LIN {X 0,Y 251.063,Z 534.012,A -85,B 0,C 180,E1 -18793.743,E2 -18793.743} C_VEL
LIN {X 0,Y 249.355,Z 538.84,A -85,B 0,C 180,E1 -18796.138,E2 -18796.138} C_VEL
LIN {X 0,Y 248.191,Z 542.574,A -85,B 0,C 180,E1 -18798.566,E2 -18798.566} C_VEL
LIN {X 0,Y 247.654,Z 544.519,A -85,B 0,C 180,E1 -18800.195,E2 -18800.195} C_VEL
LIN {X 0,Y 247.265,Z 546.047,A -85,B 0,C 180,E1 -18801.829,E2 -18801.829} C_VEL
LIN {X 0,Y 246.923,Z 547.841,A -85,B 0,C 180,E1 -18805.101,E2 -18805.101} C_VEL
LIN {X 0,Y 246.919,Z 548.165,A -85,B 0,C 180,E1 -18806.736,E2 -18806.736} C_VEL
LIN {X 0,Y 246.996,Z 548.103,A -85,B 0,C 180,E1 -18808.368,E2 -18808.368} C_VEL
LIN {X 0,Y 247.028,Z 547.606,A -85,B 0,C 180,E1 -18809.999,E2 -18809.999} C_VEL
LIN {X 0,Y 247.019,Z 546.702,A -85,B 0,C 180,E1 -18811.629,E2 -18811.629} C_VEL
LIN {X 0,Y 246.976,Z 545.393,A -85,B 0,C 180,E1 -18813.261,E2 -18813.261} C_VEL
LIN {X 0,Y 246.983,Z 543.321,A -85,B 0,C 180,E1 -18815.163,E2 -18815.163} C_VEL
LIN {X 0,Y 247.257,Z 538.751,A -85,B 0,C 180,E1 -18818.169,E2 -18818.169} C_VEL
LIN {X 0,Y 247.724,Z 533.748,A -85,B 0,C 180,E1 -18820.625,E2 -18820.625} C_VEL
LIN {X 0,Y 248.523,Z 527.438,A -85,B 0,C 180,E1 -18823.074,E2 -18823.074} C_VEL
LIN {X 0,Y 249.77,Z 519.531,A -85,B 0,C 180,E1 -18825.503,E2 -18825.503} C_VEL
LIN {X 0,Y 251.093,Z 511.441,A -85,B 0,C 180,E1 -18827.51,E2 -18827.51} C_VEL
LIN {X 0,Y 252.671,Z 501.551,A -85,B 0,C 180,E1 -18829.497,E2 -18829.497} C_VEL
LIN {X 0,Y 253.852,Z 493.137,A -85,B 0,C 180,E1 -18830.881,E2 -18830.881} C_VEL
LIN {X 0,Y 255.388,Z 483.003,A -85,B 0,C 180,E1 -18832.232,E2 -18832.232} C_VEL
LIN {X 0,Y 256.919,Z 471.105,A -85,B 0,C 180,E1 -18833.474,E2 -18833.474} C_VEL
LIN {X 0,Y 258.118,Z 458.702,A -85,B 0,C 180,E1 -18834.425,E2 -18834.425} C_VEL
LIN {X 0,Y 259.131,Z 444.941,A -85,B 0,C 180,E1 -18835.125,E2 -18835.125} C_VEL
LIN {X 0,Y 260.839,Z 386.415,A -85,B 0,C 180,E1 -18836.75,E2 -18836.75} C_VEL
LIN {X 0,Y 257.203,Z 354.534,A -85,B 0,C 180,E1 -18838.025,E2 -18838.025} C_VEL
LIN {X 0,Y 255.532,Z 344.226,A -85,B 0,C 180,E1 -18838.495,E2 -18838.495} C_VEL
LIN {X 0,Y 252.43,Z 335.333,A -85,B 0,C 180,E1 -18839.106,E2 -18839.106} C_VEL
LIN {X 0,Y 250.392,Z 325.515,A -85,B 0,C 180,E1 -18842.644,E2 -18842.644} C_VEL
LIN {X 0,Y 249.077,Z 319.458,A -85,B 0,C 180,E1 -18844.943,E2 -18844.943} C_VEL
LIN {X 0,Y 249.022,Z 319.465,A -85,B 0,C 180,E1 -18848.379,E2 -18848.379} C_VEL
LIN {X 0,Y 248.997,Z 319.468,A -85,B 0,C 180,E1 -18852.789,E2 -18852.789} C_VEL
LIN {X 0,Y 249.014,Z 319.465,A -85,B 0,C 180,E1 -18857.362,E2 -18857.362} C_VEL
LIN {X 0,Y 249.034,Z 319.461,A -85,B 0,C 180,E1 -18861.621,E2 -18861.621} C_VEL
LIN {X 0,Y 249.055,Z 319.459,A -85,B 0,C 180,E1 -18865.641,E2 -18865.641} C_VEL
LIN {X 0,Y 249.046,Z 319.461,A -85,B 0,C 180,E1 -18869.472,E2 -18869.472} C_VEL
LIN {X 0,Y 249.067,Z 319.461,A -85,B 0,C 180,E1 -18873.162,E2 -18873.162} C_VEL
LIN {X 0,Y 249.072,Z 319.458,A -85,B 0,C 180,E1 -18876.732,E2 -18876.732} C_VEL
LIN {X 0,Y 249.103,Z 319.45,A -85,B 0,C 180,E1 -18880.211,E2 -18880.211} C_VEL
LIN {X 0,Y 249.235,Z 319.428,A -85,B 0,C 180,E1 -18883.621,E2 -18883.621} C_VEL
LIN {X 0,Y 249.245,Z 319.436,A -85,B 0,C 180,E1 -18888.616,E2 -18888.616} C_VEL
LIN {X 0,Y 249.474,Z 319.398,A -85,B 0,C 180,E1 -18891.903,E2 -18891.903} C_VEL
LIN {X 0,Y 249.428,Z 319.407,A -85,B 0,C 180,E1 -18896.77,E2 -18896.77} C_VEL
LIN {X 0,Y 249.72,Z 319.377,A -85,B 0,C 180,E1 -18900,E2 -18900} C_VEL
LIN {X 0,Y 249.425,Z 319.409,A -85,B 0,C 180,E1 -18903.231,E2 -18903.231} C_VEL
LIN {X 0,Y 249.423,Z 319.397,A -85,B 0,C 180,E1 -18906.567,E2 -18906.567} C_VEL
LIN {X 0,Y 249.336,Z 319.421,A -85,B 0,C 180,E1 -18909.737,E2 -18909.737} C_VEL
LIN {X 0,Y 249.198,Z 319.438,A -85,B 0,C 180,E1 -18914.704,E2 -18914.704} C_VEL
LIN {X 0,Y 249.132,Z 319.453,A -85,B 0,C 180,E1 -18918.078,E2 -18918.078} C_VEL
LIN {X 0,Y 249.077,Z 319.454,A -85,B 0,C 180,E1 -18921.519,E2 -18921.519} C_VEL
LIN {X 0,Y 249.111,Z 319.452,A -85,B 0,C 180,E1 -18925.476,E2 -18925.476} C_VEL
LIN {X 0,Y 249.077,Z 319.455,A -85,B 0,C 180,E1 -18928.994,E2 -18928.994} C_VEL
LIN {X 0,Y 249.025,Z 319.464,A -85,B 0,C 180,E1 -18932.427,E2 -18932.427} C_VEL
LIN {X 0,Y 249.041,Z 319.462,A -85,B 0,C 180,E1 -18936.344,E2 -18936.344} C_VEL
LIN {X 0,Y 248.973,Z 319.469,A -85,B 0,C 180,E1 -18940.485,E2 -18940.485} C_VEL
LIN {X 0,Y 248.957,Z 319.471,A -85,B 0,C 180,E1 -18944.89,E2 -18944.89} C_VEL
LIN {X 0,Y 248.975,Z 319.469,A -85,B 0,C 180,E1 -18947.356,E2 -18947.356} C_VEL
LIN {X 0,Y 249.038,Z 319.461,A -85,B 0,C 180,E1 -18952.203,E2 -18952.203} C_VEL
LIN {X 0,Y 249.04,Z 319.462,A -85,B 0,C 180,E1 -18955.641,E2 -18955.641} C_VEL
LIN {X 0,Y 249,Z 319.468,A -85,B 0,C 180,E1 -18959.468,E2 -18959.468} C_VEL
LIN {X 0,Y 249.033,Z 319.465,A -85,B 0,C 180,E1 -18963.159,E2 -18963.159} C_VEL
LIN {X 0,Y 249.053,Z 319.461,A -85,B 0,C 180,E1 -18966.732,E2 -18966.732} C_VEL
LIN {X 0,Y 249.085,Z 319.458,A -85,B 0,C 180,E1 -18970.211,E2 -18970.211} C_VEL
LIN {X 0,Y 249.248,Z 319.437,A -85,B 0,C 180,E1 -18974.695,E2 -18974.695} C_VEL
LIN {X 0,Y 250.36,Z 322.47,A -85,B 0,C 180,E1 -18974.92,E2 -18974.92} C_VEL
LIN {X 0,Y 255.478,Z 334.885,A -85,B 0,C 180,E1 -18975.815,E2 -18975.815} C_VEL
LIN {X 0,Y 261.05,Z 350.896,A -85,B 0,C 180,E1 -18976.822,E2 -18976.822} C_VEL
LIN {X 0,Y 261.764,Z 354.425,A -85,B 0,C 180,E1 -18976.99,E2 -18976.99} C_VEL
LIN {X 0,Y 259.347,Z 426.547,A -85,B 0,C 180,E1 -18978.948,E2 -18978.948} C_VEL
LIN {X 0,Y 258.556,Z 440.569,A -85,B 0,C 180,E1 -18979.676,E2 -18979.676} C_VEL
LIN {X 0,Y 257.383,Z 453.393,A -85,B 0,C 180,E1 -18980.671,E2 -18980.671} C_VEL
LIN {X 0,Y 256.154,Z 465.078,A -85,B 0,C 180,E1 -18981.918,E2 -18981.918} C_VEL
LIN {X 0,Y 254.644,Z 476.639,A -85,B 0,C 180,E1 -18983.505,E2 -18983.505} C_VEL
LIN {X 0,Y 253.095,Z 486.581,A -85,B 0,C 180,E1 -18985.223,E2 -18985.223} C_VEL
LIN {X 0,Y 251.502,Z 495.769,A -85,B 0,C 180,E1 -18987.198,E2 -18987.198} C_VEL
LIN {X 0,Y 250.012,Z 504.701,A -85,B 0,C 180,E1 -18989.599,E2 -18989.599} C_VEL
LIN {X 0,Y 248.864,Z 511.881,A -85,B 0,C 180,E1 -18992.024,E2 -18992.024} C_VEL
LIN {X 0,Y 247.927,Z 518.411,A -85,B 0,C 180,E1 -18994.88,E2 -18994.88} C_VEL
LIN {X 0,Y 247.376,Z 522.735,A -85,B 0,C 180,E1 -18997.346,E2 -18997.346} C_VEL
LIN {X 0,Y 246.917,Z 525.994,A -85,B 0,C 180,E1 -18999.834,E2 -18999.834} C_VEL
LIN {X 0,Y 246.776,Z 527.616,A -85,B 0,C 180,E1 -19001.5,E2 -19001.5} C_VEL
LIN {X 0,Y 246.791,Z 529.434,A -85,B 0,C 180,E1 -19004.479,E2 -19004.479} C_VEL
LIN {X 0,Y 246.83,Z 529.9,A -85,B 0,C 180,E1 -19006.544,E2 -19006.544} C_VEL
LIN {X 0,Y 247.068,Z 529.849,A -85,B 0,C 180,E1 -19008.235,E2 -19008.235} C_VEL
LIN {X 0,Y 247.581,Z 529.079,A -85,B 0,C 180,E1 -19010.485,E2 -19010.485} C_VEL
LIN {X 0,Y 248.484,Z 527.059,A -85,B 0,C 180,E1 -19013.327,E2 -19013.327} C_VEL
LIN {X 0,Y 249.626,Z 524.337,A -85,B 0,C 180,E1 -19015.719,E2 -19015.719} C_VEL
LIN {X 0,Y 251.27,Z 520.117,A -85,B 0,C 180,E1 -19018.392,E2 -19018.392} C_VEL
LIN {X 0,Y 253.306,Z 514.524,A -85,B 0,C 180,E1 -19021.018,E2 -19021.018} C_VEL
LIN {X 0,Y 255.581,Z 508.057,A -85,B 0,C 180,E1 -19023.365,E2 -19023.365} C_VEL
LIN {X 0,Y 258.262,Z 499.864,A -85,B 0,C 180,E1 -19025.713,E2 -19025.713} C_VEL
LIN {X 0,Y 261.05,Z 490.753,A -85,B 0,C 180,E1 -19027.77,E2 -19027.77} C_VEL
LIN {X 0,Y 264.031,Z 479.746,A -85,B 0,C 180,E1 -19029.706,E2 -19029.706} C_VEL
LIN {X 0,Y 266.539,Z 468.701,A -85,B 0,C 180,E1 -19031.239,E2 -19031.239} C_VEL
LIN {X 0,Y 268.671,Z 457.188,A -85,B 0,C 180,E1 -19032.471,E2 -19032.471} C_VEL
LIN {X 0,Y 270.514,Z 444.524,A -85,B 0,C 180,E1 -19033.482,E2 -19033.482} C_VEL
LIN {X 0,Y 271.823,Z 431.405,A -85,B 0,C 180,E1 -19034.215,E2 -19034.215} C_VEL
LIN {X 0,Y 272.675,Z 416.434,A -85,B 0,C 180,E1 -19034.695,E2 -19034.695} C_VEL
LIN {X 0,Y 274.89,Z 366.849,A -85,B 0,C 180,E1 -19035.961,E2 -19035.961} C_VEL
LIN {X 0,Y 268.89,Z 353.904,A -85,B 0,C 180,E1 -19037.381,E2 -19037.381} C_VEL
LIN {X 0,Y 260.051,Z 337.508,A -85,B 0,C 180,E1 -19039.563,E2 -19039.563} C_VEL
LIN {X 0,Y 253.907,Z 327.715,A -85,B 0,C 180,E1 -19041.162,E2 -19041.162} C_VEL
LIN {X 0,Y 251.471,Z 323.932,A -85,B 0,C 180,E1 -19041.827,E2 -19041.827} C_VEL
LIN {X 0,Y 249.688,Z 321.608,A -85,B 0,C 180,E1 -19042.308,E2 -19042.308} C_VEL
LIN {X 0,Y 249.177,Z 320.079,A -85,B 0,C 180,E1 -19042.516,E2 -19042.516} C_VEL
LIN {X 0,Y 249.108,Z 319.459,A -85,B 0,C 180,E1 -19042.838,E2 -19042.838} C_VEL
LIN {X 0,Y 249.034,Z 319.461,A -85,B 0,C 180,E1 -19047.574,E2 -19047.574} C_VEL
LIN {X 0,Y 249.1,Z 319.457,A -85,B 0,C 180,E1 -19051.338,E2 -19051.338} C_VEL
LIN {X 0,Y 249.154,Z 319.45,A -85,B 0,C 180,E1 -19054.969,E2 -19054.969} C_VEL
LIN {X 0,Y 249.113,Z 319.446,A -85,B 0,C 180,E1 -19060.212,E2 -19060.212} C_VEL
LIN {X 0,Y 249.245,Z 319.437,A -85,B 0,C 180,E1 -19063.622,E2 -19063.622} C_VEL
LIN {X 0,Y 249.255,Z 319.436,A -85,B 0,C 180,E1 -19068.617,E2 -19068.617} C_VEL
LIN {X 0,Y 249.484,Z 319.4,A -85,B 0,C 180,E1 -19071.903,E2 -19071.903} C_VEL
LIN {X 0,Y 249.435,Z 319.403,A -85,B 0,C 180,E1 -19076.769,E2 -19076.769} C_VEL
LIN {X 0,Y 249.723,Z 319.363,A -85,B 0,C 180,E1 -19080,E2 -19080} C_VEL
LIN {X 0,Y 249.437,Z 319.41,A -85,B 0,C 180,E1 -19083.23,E2 -19083.23} C_VEL
LIN {X 0,Y 249.445,Z 319.395,A -85,B 0,C 180,E1 -19086.358,E2 -19086.358} C_VEL
LIN {X 0,Y 248.906,Z 319.472,A -85,B 0,C 180,E1 -19087.704,E2 -19087.704} C_VEL
LIN {X 0,Y 247.33,Z 319.675,A -85,B 0,C 180,E1 -19089.024,E2 -19089.024} C_VEL
LIN {X 0,Y 243.425,Z 320.169,A -85,B 0,C 180,E1 -19091.678,E2 -19091.678} C_VEL
LIN {X 0,Y 242.273,Z 320.307,A -85,B 0,C 180,E1 -19093.067,E2 -19093.067} C_VEL
LIN {X 0,Y 242.162,Z 320.316,A -85,B 0,C 180,E1 -19093.539,E2 -19093.539} C_VEL
LIN {X 0,Y 242.153,Z 320.307,A -85,B 0,C 180,E1 -19096.872,E2 -19096.872} C_VEL
LIN {X 0,Y 242.029,Z 320.324,A -85,B 0,C 180,E1 -19101.686,E2 -19101.686} C_VEL
LIN {X 0,Y 242.069,Z 320.318,A -85,B 0,C 180,E1 -19105.838,E2 -19105.838} C_VEL
LIN {X 0,Y 242.033,Z 320.324,A -85,B 0,C 180,E1 -19109.58,E2 -19109.58} C_VEL
LIN {X 0,Y 241.983,Z 320.332,A -85,B 0,C 180,E1 -19113.492,E2 -19113.492} C_VEL
LIN {X 0,Y 241.992,Z 320.333,A -85,B 0,C 180,E1 -19117.582,E2 -19117.582} C_VEL
LIN {X 0,Y 241.936,Z 320.351,A -85,B 0,C 180,E1 -19121.923,E2 -19121.923} C_VEL
LIN {X 0,Y 241.936,Z 320.499,A -85,B 0,C 180,E1 -19124.086,E2 -19124.086} C_VEL
LIN {X 0,Y 244.233,Z 327.949,A -85,B 0,C 180,E1 -19128.121,E2 -19128.121} C_VEL
LIN {X 0,Y 245.847,Z 333.529,A -85,B 0,C 180,E1 -19130.843,E2 -19130.843} C_VEL
LIN {X 0,Y 248.328,Z 337.884,A -85,B 0,C 180,E1 -19131.574,E2 -19131.574} C_VEL
LIN {X 0,Y 254.341,Z 348.606,A -85,B 0,C 180,E1 -19133.258,E2 -19133.258} C_VEL
LIN {X 0,Y 261.31,Z 362.634,A -85,B 0,C 180,E1 -19135.116,E2 -19135.116} C_VEL
LIN {X 0,Y 265.318,Z 371.754,A -85,B 0,C 180,E1 -19136.15,E2 -19136.15} C_VEL
LIN {X 0,Y 268.268,Z 390.386,A -85,B 0,C 180,E1 -19137.283,E2 -19137.283} C_VEL
LIN {X 0,Y 265.892,Z 443.094,A -85,B 0,C 180,E1 -19138.704,E2 -19138.704} C_VEL
LIN {X 0,Y 264.543,Z 456.576,A -85,B 0,C 180,E1 -19139.333,E2 -19139.333} C_VEL
LIN {X 0,Y 262.561,Z 469.325,A -85,B 0,C 180,E1 -19140.206,E2 -19140.206} C_VEL
LIN {X 0,Y 260.161,Z 481.261,A -85,B 0,C 180,E1 -19141.346,E2 -19141.346} C_VEL
LIN {X 0,Y 257.375,Z 492.686,A -85,B 0,C 180,E1 -19142.781,E2 -19142.781} C_VEL
LIN {X 0,Y 254.574,Z 502.997,A -85,B 0,C 180,E1 -19144.445,E2 -19144.445} C_VEL
LIN {X 0,Y 251.89,Z 511.459,A -85,B 0,C 180,E1 -19146.135,E2 -19146.135} C_VEL
LIN {X 0,Y 248.808,Z 520.659,A -85,B 0,C 180,E1 -19148.456,E2 -19148.456} C_VEL
LIN {X 0,Y 246.34,Z 528.074,A -85,B 0,C 180,E1 -19150.846,E2 -19150.846} C_VEL
LIN {X 0,Y 244.26,Z 534.062,A -85,B 0,C 180,E1 -19153.277,E2 -19153.277} C_VEL
LIN {X 0,Y 242.433,Z 538.823,A -85,B 0,C 180,E1 -19155.734,E2 -19155.734} C_VEL
LIN {X 0,Y 241.217,Z 542.494,A -85,B 0,C 180,E1 -19158.231,E2 -19158.231} C_VEL
LIN {X 0,Y 240.641,Z 544.408,A -85,B 0,C 180,E1 -19159.907,E2 -19159.907} C_VEL
LIN {X 0,Y 240.215,Z 545.881,A -85,B 0,C 180,E1 -19161.587,E2 -19161.587} C_VEL
LIN {X 0,Y 239.845,Z 547.617,A -85,B 0,C 180,E1 -19164.956,E2 -19164.956} C_VEL
LIN {X 0,Y 239.821,Z 547.913,A -85,B 0,C 180,E1 -19166.639,E2 -19166.639} C_VEL
LIN {X 0,Y 239.902,Z 547.807,A -85,B 0,C 180,E1 -19168.32,E2 -19168.32} C_VEL
LIN {X 0,Y 239.957,Z 547.272,A -85,B 0,C 180,E1 -19169.999,E2 -19169.999} C_VEL
LIN {X 0,Y 239.949,Z 546.34,A -85,B 0,C 180,E1 -19171.677,E2 -19171.677} C_VEL
LIN {X 0,Y 239.876,Z 545,A -85,B 0,C 180,E1 -19173.358,E2 -19173.358} C_VEL
LIN {X 0,Y 239.919,Z 542.144,A -85,B 0,C 180,E1 -19175.883,E2 -19175.883} C_VEL
LIN {X 0,Y 240.197,Z 538.234,A -85,B 0,C 180,E1 -19178.411,E2 -19178.411} C_VEL
LIN {X 0,Y 240.703,Z 533.162,A -85,B 0,C 180,E1 -19180.939,E2 -19180.939} C_VEL
LIN {X 0,Y 241.577,Z 526.769,A -85,B 0,C 180,E1 -19183.457,E2 -19183.457} C_VEL
LIN {X 0,Y 242.873,Z 518.738,A -85,B 0,C 180,E1 -19185.955,E2 -19185.955} C_VEL
LIN {X 0,Y 244.141,Z 511.311,A -85,B 0,C 180,E1 -19187.841,E2 -19187.841} C_VEL
LIN {X 0,Y 245.738,Z 501.719,A -85,B 0,C 180,E1 -19189.83,E2 -19189.83} C_VEL
LIN {X 0,Y 246.977,Z 493.264,A -85,B 0,C 180,E1 -19191.272,E2 -19191.272} C_VEL
LIN {X 0,Y 248.785,Z 481.618,A -85,B 0,C 180,E1 -19192.855,E2 -19192.855} C_VEL
LIN {X 0,Y 250.355,Z 469.287,A -85,B 0,C 180,E1 -19194.128,E2 -19194.128} C_VEL
LIN {X 0,Y 251.652,Z 456.296,A -85,B 0,C 180,E1 -19195.095,E2 -19195.095} C_VEL
LIN {X 0,Y 252.543,Z 443.755,A -85,B 0,C 180,E1 -19195.717,E2 -19195.717} C_VEL
LIN {X 0,Y 254.155,Z 384.923,A -85,B 0,C 180,E1 -19197.39,E2 -19197.39} C_VEL
LIN {X 0,Y 249.791,Z 349.447,A -85,B 0,C 180,E1 -19198.899,E2 -19198.899} C_VEL
LIN {X 0,Y 248.836,Z 345.277,A -85,B 0,C 180,E1 -19199.125,E2 -19199.125} C_VEL
LIN {X 0,Y 245.191,Z 335.113,A -85,B 0,C 180,E1 -19199.838,E2 -19199.838} C_VEL
LIN {X 0,Y 242.941,Z 324.443,A -85,B 0,C 180,E1 -19203.838,E2 -19203.838} C_VEL
LIN {X 0,Y 242.001,Z 320.339,A -85,B 0,C 180,E1 -19205.506,E2 -19205.506} C_VEL
LIN {X 0,Y 241.953,Z 320.343,A -85,B 0,C 180,E1 -19209.718,E2 -19209.718} C_VEL
LIN {X 0,Y 241.919,Z 320.351,A -85,B 0,C 180,E1 -19214.202,E2 -19214.202} C_VEL
LIN {X 0,Y 241.94,Z 320.348,A -85,B 0,C 180,E1 -19218.078,E2 -19218.078} C_VEL
LIN {X 0,Y 241.998,Z 320.34,A -85,B 0,C 180,E1 -19222.42,E2 -19222.42} C_VEL
LIN {X 0,Y 241.985,Z 320.342,A -85,B 0,C 180,E1 -19226.508,E2 -19226.508} C_VEL
LIN {X 0,Y 242.031,Z 320.336,A -85,B 0,C 180,E1 -19230.586,E2 -19230.586} C_VEL
LIN {X 0,Y 242.061,Z 320.33,A -85,B 0,C 180,E1 -19234.182,E2 -19234.182} C_VEL
LIN {X 0,Y 242.046,Z 320.333,A -85,B 0,C 180,E1 -19238.297,E2 -19238.297} C_VEL
LIN {X 0,Y 242.156,Z 320.306,A -85,B 0,C 180,E1 -19243.278,E2 -19243.278} C_VEL
LIN {X 0,Y 242.178,Z 320.316,A -85,B 0,C 180,E1 -19248.279,E2 -19248.279} C_VEL
LIN {X 0,Y 242.42,Z 320.278,A -85,B 0,C 180,E1 -19251.665,E2 -19251.665} C_VEL
LIN {X 0,Y 242.251,Z 320.291,A -85,B 0,C 180,E1 -19255.007,E2 -19255.007} C_VEL
LIN {X 0,Y 242.629,Z 320.259,A -85,B 0,C 180,E1 -19258.34,E2 -19258.34} C_VEL
LIN {X 0,Y 242.628,Z 320.26,A -85,B 0,C 180,E1 -19261.66,E2 -19261.66} C_VEL
LIN {X 0,Y 242.4,Z 320.271,A -85,B 0,C 180,E1 -19266.66,E2 -19266.66} C_VEL
LIN {X 0,Y 242.26,Z 320.304,A -85,B 0,C 180,E1 -19270.024,E2 -19270.024} C_VEL
LIN {X 0,Y 242.16,Z 320.314,A -85,B 0,C 180,E1 -19275.141,E2 -19275.141} C_VEL
LIN {X 0,Y 242.066,Z 320.331,A -85,B 0,C 180,E1 -19278.625,E2 -19278.625} C_VEL
LIN {X 0,Y 242,Z 320.337,A -85,B 0,C 180,E1 -19282.181,E2 -19282.181} C_VEL
LIN {X 0,Y 242.061,Z 320.331,A -85,B 0,C 180,E1 -19285.839,E2 -19285.839} C_VEL
LIN {X 0,Y 242.025,Z 320.333,A -85,B 0,C 180,E1 -19289.581,E2 -19289.581} C_VEL
LIN {X 0,Y 241.975,Z 320.336,A -85,B 0,C 180,E1 -19293.494,E2 -19293.494} C_VEL
LIN {X 0,Y 241.982,Z 320.338,A -85,B 0,C 180,E1 -19297.584,E2 -19297.584} C_VEL
LIN {X 0,Y 241.903,Z 320.349,A -85,B 0,C 180,E1 -19301.93,E2 -19301.93} C_VEL
LIN {X 0,Y 241.896,Z 320.353,A -85,B 0,C 180,E1 -19306.581,E2 -19306.581} C_VEL
LIN {X 0,Y 241.989,Z 320.34,A -85,B 0,C 180,E1 -19311.643,E2 -19311.643} C_VEL
LIN {X 0,Y 241.977,Z 320.342,A -85,B 0,C 180,E1 -19314.489,E2 -19314.489} C_VEL
LIN {X 0,Y 241.95,Z 320.345,A -85,B 0,C 180,E1 -19318.478,E2 -19318.478} C_VEL
LIN {X 0,Y 241.966,Z 320.343,A -85,B 0,C 180,E1 -19322.309,E2 -19322.309} C_VEL
LIN {X 0,Y 242.023,Z 320.337,A -85,B 0,C 180,E1 -19326.014,E2 -19326.014} C_VEL
LIN {X 0,Y 242.02,Z 320.336,A -85,B 0,C 180,E1 -19329.608,E2 -19329.608} C_VEL
LIN {X 0,Y 242.165,Z 320.397,A -85,B 0,C 180,E1 -19333.974,E2 -19333.974} C_VEL
LIN {X 0,Y 243.252,Z 323.281,A -85,B 0,C 180,E1 -19334.187,E2 -19334.187} C_VEL
LIN {X 0,Y 247.71,Z 333.288,A -85,B 0,C 180,E1 -19334.983,E2 -19334.983} C_VEL
LIN {X 0,Y 254.637,Z 352.807,A -85,B 0,C 180,E1 -19336.279,E2 -19336.279} C_VEL
LIN {X 0,Y 255.173,Z 355.269,A -85,B 0,C 180,E1 -19336.405,E2 -19336.405} C_VEL
LIN {X 0,Y 252.769,Z 426.097,A -85,B 0,C 180,E1 -19338.367,E2 -19338.367} C_VEL
LIN {X 0,Y 251.992,Z 439.389,A -85,B 0,C 180,E1 -19339.049,E2 -19339.049} C_VEL
LIN {X 0,Y 250.825,Z 452.119,A -85,B 0,C 180,E1 -19340.017,E2 -19340.017} C_VEL
LIN {X 0,Y 249.515,Z 464.201,A -85,B 0,C 180,E1 -19341.293,E2 -19341.293} C_VEL
LIN {X 0,Y 248.126,Z 474.723,A -85,B 0,C 180,E1 -19342.728,E2 -19342.728} C_VEL
LIN {X 0,Y 246.484,Z 485.026,A -85,B 0,C 180,E1 -19344.479,E2 -19344.479} C_VEL
LIN {X 0,Y 245.015,Z 493.699,A -85,B 0,C 180,E1 -19346.301,E2 -19346.301} C_VEL
LIN {X 0,Y 243.608,Z 501.688,A -85,B 0,C 180,E1 -19348.348,E2 -19348.348} C_VEL
LIN {X 0,Y 242.236,Z 509.503,A -85,B 0,C 180,E1 -19350.832,E2 -19350.832} C_VEL
LIN {X 0,Y 241.248,Z 515.75,A -85,B 0,C 180,E1 -19353.341,E2 -19353.341} C_VEL
LIN {X 0,Y 240.629,Z 520.473,A -85,B 0,C 180,E1 -19355.728,E2 -19355.728} C_VEL
LIN {X 0,Y 240.057,Z 524.561,A -85,B 0,C 180,E1 -19358.418,E2 -19358.418} C_VEL
LIN {X 0,Y 239.798,Z 526.552,A -85,B 0,C 180,E1 -19360.129,E2 -19360.129} C_VEL
LIN {X 0,Y 239.681,Z 528.111,A -85,B 0,C 180,E1 -19361.846,E2 -19361.846} C_VEL
LIN {X 0,Y 239.713,Z 529.702,A -85,B 0,C 180,E1 -19364.644,E2 -19364.644} C_VEL
LIN {X 0,Y 239.783,Z 530.199,A -85,B 0,C 180,E1 -19367.045,E2 -19367.045} C_VEL
LIN {X 0,Y 240.07,Z 530.059,A -85,B 0,C 180,E1 -19368.786,E2 -19368.786} C_VEL
LIN {X 0,Y 240.571,Z 529.358,A -85,B 0,C 180,E1 -19370.796,E2 -19370.796} C_VEL
LIN {X 0,Y 241.666,Z 527.077,A -85,B 0,C 180,E1 -19374.026,E2 -19374.026} C_VEL
LIN {X 0,Y 242.767,Z 524.638,A -85,B 0,C 180,E1 -19376.176,E2 -19376.176} C_VEL
LIN {X 0,Y 244.7,Z 519.876,A -85,B 0,C 180,E1 -19379.227,E2 -19379.227} C_VEL
LIN {X 0,Y 247.211,Z 513.382,A -85,B 0,C 180,E1 -19382.212,E2 -19382.212} C_VEL
LIN {X 0,Y 249.795,Z 506.389,A -85,B 0,C 180,E1 -19384.672,E2 -19384.672} C_VEL
LIN {X 0,Y 252.323,Z 498.812,A -85,B 0,C 180,E1 -19386.788,E2 -19386.788} C_VEL
LIN {X 0,Y 255.489,Z 488.727,A -85,B 0,C 180,E1 -19388.995,E2 -19388.995} C_VEL
LIN {X 0,Y 258.373,Z 478.487,A -85,B 0,C 180,E1 -19390.756,E2 -19390.756} C_VEL
LIN {X 0,Y 260.973,Z 466.927,A -85,B 0,C 180,E1 -19392.319,E2 -19392.319} C_VEL
LIN {X 0,Y 263.246,Z 454.87,A -85,B 0,C 180,E1 -19393.562,E2 -19393.562} C_VEL
LIN {X 0,Y 265.009,Z 442.377,A -85,B 0,C 180,E1 -19394.517,E2 -19394.517} C_VEL
LIN {X 0,Y 266.236,Z 429.336,A -85,B 0,C 180,E1 -19395.192,E2 -19395.192} C_VEL
LIN {X 0,Y 267.289,Z 411.227,A -85,B 0,C 180,E1 -19395.715,E2 -19395.715} C_VEL
LIN {X 0,Y 269.108,Z 368.812,A -85,B 0,C 180,E1 -19396.84,E2 -19396.84} C_VEL
LIN {X 0,Y 262.767,Z 355.414,A -85,B 0,C 180,E1 -19398.411,E2 -19398.411} C_VEL
LIN {X 0,Y 255.455,Z 341.823,A -85,B 0,C 180,E1 -19400.309,E2 -19400.309} C_VEL
LIN {X 0,Y 249.505,Z 332.272,A -85,B 0,C 180,E1 -19401.926,E2 -19401.926} C_VEL
LIN {X 0,Y 247.267,Z 328.916,A -85,B 0,C 180,E1 -19402.556,E2 -19402.556} C_VEL
LIN {X 0,Y 245.28,Z 325.85,A -85,B 0,C 180,E1 -19403.136,E2 -19403.136} C_VEL
LIN {X 0,Y 244.295,Z 324.728,A -85,B 0,C 180,E1 -19403.413,E2 -19403.413} C_VEL
LIN {X 0,Y 242.626,Z 322.509,A -85,B 0,C 180,E1 -19403.904,E2 -19403.904} C_VEL
LIN {X 0,Y 242.017,Z 320.466,A -85,B 0,C 180,E1 -19404.175,E2 -19404.175} C_VEL
LIN {X 0,Y 241.978,Z 320.345,A -85,B 0,C 180,E1 -19408.48,E2 -19408.48} C_VEL
LIN {X 0,Y 242.012,Z 320.335,A -85,B 0,C 180,E1 -19412.313,E2 -19412.313} C_VEL
LIN {X 0,Y 242.06,Z 320.327,A -85,B 0,C 180,E1 -19416.016,E2 -19416.016} C_VEL
LIN {X 0,Y 242.04,Z 320.332,A -85,B 0,C 180,E1 -19419.608,E2 -19419.608} C_VEL
LIN {X 0,Y 242.166,Z 320.32,A -85,B 0,C 180,E1 -19423.278,E2 -19423.278} C_VEL
LIN {X 0,Y 242.189,Z 320.316,A -85,B 0,C 180,E1 -19428.28,E2 -19428.28} C_VEL
LIN {X 0,Y 242.43,Z 320.276,A -85,B 0,C 180,E1 -19431.666,E2 -19431.666} C_VEL
LIN {X 0,Y 242.259,Z 320.294,A -85,B 0,C 180,E1 -19435.007,E2 -19435.007} C_VEL
LIN {X 0,Y 242.637,Z 320.26,A -85,B 0,C 180,E1 -19438.34,E2 -19438.34} C_VEL
LIN {X 0,Y 242.638,Z 320.243,A -85,B 0,C 180,E1 -19441.66,E2 -19441.66} C_VEL
LIN {X 0,Y 242.436,Z 320.269,A -85,B 0,C 180,E1 -19446.659,E2 -19446.659} C_VEL
LIN {X 0,Y 242.348,Z 320.284,A -85,B 0,C 180,E1 -19450.02,E2 -19450.02} C_VEL
LIN {X 0,Y 242.162,Z 320.316,A -85,B 0,C 180,E1 -19453.539,E2 -19453.539} C_VEL
LIN {X 0,Y 241.428,Z 320.404,A -85,B 0,C 180,E1 -19454.926,E2 -19454.926} C_VEL
LIN {X 0,Y 238.489,Z 320.765,A -85,B 0,C 180,E1 -19457.186,E2 -19457.186} C_VEL
LIN {X 0,Y 236.053,Z 321.08,A -85,B 0,C 180,E1 -19459.028,E2 -19459.028} C_VEL
LIN {X 0,Y 235.054,Z 321.193,A -85,B 0,C 180,E1 -19460.459,E2 -19460.459} C_VEL
LIN {X 0,Y 234.996,Z 321.198,A -85,B 0,C 180,E1 -19460.944,E2 -19460.944} C_VEL
LIN {X 0,Y 234.997,Z 321.2,A -85,B 0,C 180,E1 -19466.206,E2 -19466.206} C_VEL
LIN {X 0,Y 234.934,Z 321.209,A -85,B 0,C 180,E1 -19470.567,E2 -19470.567} C_VEL
LIN {X 0,Y 234.933,Z 321.212,A -85,B 0,C 180,E1 -19474.638,E2 -19474.638} C_VEL
LIN {X 0,Y 234.944,Z 321.22,A -85,B 0,C 180,E1 -19478.944,E2 -19478.944} C_VEL
LIN {X 0,Y 234.909,Z 321.433,A -85,B 0,C 180,E1 -19482.577,E2 -19482.577} C_VEL
LIN {X 0,Y 237.376,Z 329.255,A -85,B 0,C 180,E1 -19487.08,E2 -19487.08} C_VEL
LIN {X 0,Y 238.5,Z 333.251,A -85,B 0,C 180,E1 -19489.071,E2 -19489.071} C_VEL
LIN {X 0,Y 241.379,Z 338,A -85,B 0,C 180,E1 -19489.983,E2 -19489.983} C_VEL
LIN {X 0,Y 247.642,Z 348.829,A -85,B 0,C 180,E1 -19491.858,E2 -19491.858} C_VEL
LIN {X 0,Y 255.057,Z 363.424,A -85,B 0,C 180,E1 -19493.955,E2 -19493.955} C_VEL
LIN {X 0,Y 259.996,Z 374.477,A -85,B 0,C 180,E1 -19495.296,E2 -19495.296} C_VEL
LIN {X 0,Y 262.692,Z 391.848,A -85,B 0,C 180,E1 -19496.389,E2 -19496.389} C_VEL
LIN {X 0,Y 260.18,Z 443.362,A -85,B 0,C 180,E1 -19497.797,E2 -19497.797} C_VEL
LIN {X 0,Y 258.682,Z 457.433,A -85,B 0,C 180,E1 -19498.479,E2 -19498.479} C_VEL
LIN {X 0,Y 256.674,Z 469.553,A -85,B 0,C 180,E1 -19499.337,E2 -19499.337} C_VEL
LIN {X 0,Y 254.002,Z 482.139,A -85,B 0,C 180,E1 -19500.585,E2 -19500.585} C_VEL
LIN {X 0,Y 251.123,Z 493.356,A -85,B 0,C 180,E1 -19502.045,E2 -19502.045} C_VEL
LIN {X 0,Y 248.228,Z 503.49,A -85,B 0,C 180,E1 -19503.743,E2 -19503.743} C_VEL
LIN {X 0,Y 245.44,Z 511.823,A -85,B 0,C 180,E1 -19505.467,E2 -19505.467} C_VEL
LIN {X 0,Y 242.209,Z 520.886,A -85,B 0,C 180,E1 -19507.838,E2 -19507.838} C_VEL
LIN {X 0,Y 239.642,Z 528.212,A -85,B 0,C 180,E1 -19510.289,E2 -19510.289} C_VEL
LIN {X 0,Y 237.457,Z 534.119,A -85,B 0,C 180,E1 -19512.783,E2 -19512.783} C_VEL
LIN {X 0,Y 235.534,Z 538.808,A -85,B 0,C 180,E1 -19515.307,E2 -19515.307} C_VEL
LIN {X 0,Y 234.254,Z 542.414,A -85,B 0,C 180,E1 -19517.876,E2 -19517.876} C_VEL
LIN {X 0,Y 233.615,Z 544.29,A -85,B 0,C 180,E1 -19519.6,E2 -19519.6} C_VEL
LIN {X 0,Y 232.89,Z 546.744,A -85,B 0,C 180,E1 -19523.066,E2 -19523.066} C_VEL
LIN {X 0,Y 232.761,Z 547.491,A -85,B 0,C 180,E1 -19525.14,E2 -19525.14} C_VEL
LIN {X 0,Y 232.811,Z 547.499,A -85,B 0,C 180,E1 -19528.269,E2 -19528.269} C_VEL
LIN {X 0,Y 232.888,Z 546.938,A -85,B 0,C 180,E1 -19529.999,E2 -19529.999} C_VEL
LIN {X 0,Y 232.856,Z 545.976,A -85,B 0,C 180,E1 -19531.728,E2 -19531.728} C_VEL
LIN {X 0,Y 232.78,Z 544.607,A -85,B 0,C 180,E1 -19533.461,E2 -19533.461} C_VEL
LIN {X 0,Y 232.84,Z 541.691,A -85,B 0,C 180,E1 -19536.063,E2 -19536.063} C_VEL
LIN {X 0,Y 233.134,Z 537.716,A -85,B 0,C 180,E1 -19538.668,E2 -19538.668} C_VEL
LIN {X 0,Y 233.809,Z 531.568,A -85,B 0,C 180,E1 -19541.705,E2 -19541.705} C_VEL
LIN {X 0,Y 234.888,Z 524.829,A -85,B 0,C 180,E1 -19544.289,E2 -19544.289} C_VEL
LIN {X 0,Y 236.339,Z 516.447,A -85,B 0,C 180,E1 -19546.853,E2 -19546.853} C_VEL
LIN {X 0,Y 237.773,Z 507.801,A -85,B 0,C 180,E1 -19548.972,E2 -19548.972} C_VEL
LIN {X 0,Y 239.494,Z 497.101,A -85,B 0,C 180,E1 -19551.067,E2 -19551.067} C_VEL
LIN {X 0,Y 241.185,Z 486.497,A -85,B 0,C 180,E1 -19552.71,E2 -19552.71} C_VEL
LIN {X 0,Y 243.018,Z 474.796,A -85,B 0,C 180,E1 -19554.108,E2 -19554.108} C_VEL
LIN {X 0,Y 244.369,Z 462.557,A -85,B 0,C 180,E1 -19555.213,E2 -19555.213} C_VEL
LIN {X 0,Y 245.549,Z 449.248,A -85,B 0,C 180,E1 -19556.049,E2 -19556.049} C_VEL
LIN {X 0,Y 246.167,Z 436.12,A -85,B 0,C 180,E1 -19556.548,E2 -19556.548} C_VEL
LIN {X 0,Y 247.596,Z 385.72,A -85,B 0,C 180,E1 -19557.985,E2 -19557.985} C_VEL
LIN {X 0,Y 243.336,Z 350.622,A -85,B 0,C 180,E1 -19559.522,E2 -19559.522} C_VEL
LIN {X 0,Y 242.34,Z 346.97,A -85,B 0,C 180,E1 -19559.745,E2 -19559.745} C_VEL
LIN {X 0,Y 237.906,Z 334.726,A -85,B 0,C 180,E1 -19560.678,E2 -19560.678} C_VEL
LIN {X 0,Y 235.501,Z 323.555,A -85,B 0,C 180,E1 -19565.047,E2 -19565.047} C_VEL
LIN {X 0,Y 234.932,Z 321.22,A -85,B 0,C 180,E1 -19566.087,E2 -19566.087} C_VEL
LIN {X 0,Y 234.938,Z 321.217,A -85,B 0,C 180,E1 -19568.943,E2 -19568.943} C_VEL
LIN {X 0,Y 234.876,Z 321.226,A -85,B 0,C 180,E1 -19573.486,E2 -19573.486} C_VEL
LIN {X 0,Y 234.882,Z 321.228,A -85,B 0,C 180,E1 -19576.513,E2 -19576.513} C_VEL
LIN {X 0,Y 234.95,Z 321.216,A -85,B 0,C 180,E1 -19581.085,E2 -19581.085} C_VEL
LIN {X 0,Y 234.955,Z 321.216,A -85,B 0,C 180,E1 -19585.366,E2 -19585.366} C_VEL
LIN {X 0,Y 234.963,Z 321.214,A -85,B 0,C 180,E1 -19590.156,E2 -19590.156} C_VEL
LIN {X 0,Y 234.988,Z 321.212,A -85,B 0,C 180,E1 -19593.793,E2 -19593.793} C_VEL
LIN {X 0,Y 235.005,Z 321.212,A -85,B 0,C 180,E1 -19598.969,E2 -19598.969} C_VEL
LIN {X 0,Y 235.089,Z 321.185,A -85,B 0,C 180,E1 -19603.059,E2 -19603.059} C_VEL
LIN {X 0,Y 235.138,Z 321.194,A -85,B 0,C 180,E1 -19607.923,E2 -19607.923} C_VEL
LIN {X 0,Y 235.369,Z 321.157,A -85,B 0,C 180,E1 -19611.414,E2 -19611.414} C_VEL
LIN {X 0,Y 235.397,Z 321.146,A -85,B 0,C 180,E1 -19613.141,E2 -19613.141} C_VEL
LIN {X 0,Y 235.588,Z 321.136,A -85,B 0,C 180,E1 -19618.291,E2 -19618.291} C_VEL
LIN {X 0,Y 235.587,Z 321.136,A -85,B 0,C 180,E1 -19621.71,E2 -19621.71} C_VEL
LIN {X 0,Y 235.351,Z 321.148,A -85,B 0,C 180,E1 -19626.86,E2 -19626.86} C_VEL
LIN {X 0,Y 235.207,Z 321.185,A -85,B 0,C 180,E1 -19630.328,E2 -19630.328} C_VEL
LIN {X 0,Y 235.107,Z 321.194,A -85,B 0,C 180,E1 -19635.607,E2 -19635.607} C_VEL
LIN {X 0,Y 235.001,Z 321.21,A -85,B 0,C 180,E1 -19639.206,E2 -19639.206} C_VEL
LIN {X 0,Y 234.946,Z 321.216,A -85,B 0,C 180,E1 -19642.885,E2 -19642.885} C_VEL
LIN {X 0,Y 234.963,Z 321.213,A -85,B 0,C 180,E1 -19646.658,E2 -19646.658} C_VEL
LIN {X 0,Y 234.926,Z 321.222,A -85,B 0,C 180,E1 -19650.569,E2 -19650.569} C_VEL
LIN {X 0,Y 234.924,Z 321.218,A -85,B 0,C 180,E1 -19654.639,E2 -19654.639} C_VEL
LIN {X 0,Y 234.906,Z 321.219,A -85,B 0,C 180,E1 -19658.936,E2 -19658.936} C_VEL
LIN {X 0,Y 234.848,Z 321.225,A -85,B 0,C 180,E1 -19663.495,E2 -19663.495} C_VEL
LIN {X 0,Y 234.849,Z 321.23,A -85,B 0,C 180,E1 -19666.508,E2 -19666.508} C_VEL
LIN {X 0,Y 234.914,Z 321.225,A -85,B 0,C 180,E1 -19671.08,E2 -19671.08} C_VEL
LIN {X 0,Y 234.923,Z 321.222,A -85,B 0,C 180,E1 -19675.363,E2 -19675.363} C_VEL
LIN {X 0,Y 234.897,Z 321.224,A -85,B 0,C 180,E1 -19679.429,E2 -19679.429} C_VEL
LIN {X 0,Y 234.967,Z 321.217,A -85,B 0,C 180,E1 -19683.808,E2 -19683.808} C_VEL
LIN {X 0,Y 234.989,Z 321.208,A -85,B 0,C 180,E1 -19688.969,E2 -19688.969} C_VEL
LIN {X 0,Y 235.069,Z 321.205,A -85,B 0,C 180,E1 -19693.18,E2 -19693.18} C_VEL
LIN {X 0,Y 236.2,Z 324.24,A -85,B 0,C 180,E1 -19693.421,E2 -19693.421} C_VEL
LIN {X 0,Y 241.44,Z 335.546,A -85,B 0,C 180,E1 -19694.387,E2 -19694.387} C_VEL
LIN {X 0,Y 248.137,Z 354.493,A -85,B 0,C 180,E1 -19695.693,E2 -19695.693} C_VEL
LIN {X 0,Y 248.584,Z 356.803,A -85,B 0,C 180,E1 -19695.81,E2 -19695.81} C_VEL
LIN {X 0,Y 246.156,Z 426.442,A -85,B 0,C 180,E1 -19697.788,E2 -19697.788} C_VEL
LIN {X 0,Y 245.338,Z 439.723,A -85,B 0,C 180,E1 -19698.486,E2 -19698.486} C_VEL
LIN {X 0,Y 244.068,Z 452.995,A -85,B 0,C 180,E1 -19699.529,E2 -19699.529} C_VEL
LIN {X 0,Y 242.718,Z 464.896,A -85,B 0,C 180,E1 -19700.838,E2 -19700.838} C_VEL
LIN {X 0,Y 241.106,Z 476.626,A -85,B 0,C 180,E1 -19702.515,E2 -19702.515} C_VEL
LIN {X 0,Y 239.443,Z 486.644,A -85,B 0,C 180,E1 -19704.316,E2 -19704.316} C_VEL
LIN {X 0,Y 237.9,Z 495.094,A -85,B 0,C 180,E1 -19706.19,E2 -19706.19} C_VEL
LIN {X 0,Y 236.241,Z 504.235,A -85,B 0,C 180,E1 -19708.723,E2 -19708.723} C_VEL
LIN {X 0,Y 234.923,Z 511.605,A -85,B 0,C 180,E1 -19711.287,E2 -19711.287} C_VEL
LIN {X 0,Y 234.096,Z 516.597,A -85,B 0,C 180,E1 -19713.444,E2 -19713.444} C_VEL
LIN {X 0,Y 233.389,Z 522.052,A -85,B 0,C 180,E1 -19716.42,E2 -19716.42} C_VEL
LIN {X 0,Y 232.906,Z 525.175,A -85,B 0,C 180,E1 -19718.679,E2 -19718.679} C_VEL
LIN {X 0,Y 232.679,Z 527.109,A -85,B 0,C 180,E1 -19720.442,E2 -19720.442} C_VEL
LIN {X 0,Y 232.571,Z 528.568,A -85,B 0,C 180,E1 -19722.213,E2 -19722.213} C_VEL
LIN {X 0,Y 232.619,Z 529.966,A -85,B 0,C 180,E1 -19724.804,E2 -19724.804} C_VEL
LIN {X 0,Y 232.772,Z 530.479,A -85,B 0,C 180,E1 -19727.574,E2 -19727.574} C_VEL
LIN {X 0,Y 233.105,Z 530.252,A -85,B 0,C 180,E1 -19729.37,E2 -19729.37} C_VEL
LIN {X 0,Y 233.584,Z 529.621,A -85,B 0,C 180,E1 -19731.166,E2 -19731.166} C_VEL
LIN {X 0,Y 234.147,Z 528.581,A -85,B 0,C 180,E1 -19732.968,E2 -19732.968} C_VEL
LIN {X 0,Y 234.892,Z 527.057,A -85,B 0,C 180,E1 -19734.765,E2 -19734.765} C_VEL
LIN {X 0,Y 236.302,Z 524.042,A -85,B 0,C 180,E1 -19737.356,E2 -19737.356} C_VEL
LIN {X 0,Y 238.21,Z 519.62,A -85,B 0,C 180,E1 -19740.104,E2 -19740.104} C_VEL
LIN {X 0,Y 240.5,Z 514.038,A -85,B 0,C 180,E1 -19742.727,E2 -19742.727} C_VEL
LIN {X 0,Y 243.244,Z 506.978,A -85,B 0,C 180,E1 -19745.301,E2 -19745.301} C_VEL
LIN {X 0,Y 245.845,Z 499.689,A -85,B 0,C 180,E1 -19747.408,E2 -19747.408} C_VEL
LIN {X 0,Y 249.12,Z 489.755,A -85,B 0,C 180,E1 -19749.665,E2 -19749.665} C_VEL
LIN {X 0,Y 252.305,Z 478.96,A -85,B 0,C 180,E1 -19751.575,E2 -19751.575} C_VEL
LIN {X 0,Y 254.815,Z 468.435,A -85,B 0,C 180,E1 -19753.05,E2 -19753.05} C_VEL
LIN {X 0,Y 257.152,Z 456.692,A -85,B 0,C 180,E1 -19754.318,E2 -19754.318} C_VEL
LIN {X 0,Y 259.024,Z 444.791,A -85,B 0,C 180,E1 -19755.278,E2 -19755.278} C_VEL
LIN {X 0,Y 260.374,Z 432.054,A -85,B 0,C 180,E1 -19756.014,E2 -19756.014} C_VEL
LIN {X 0,Y 261.298,Z 417.418,A -85,B 0,C 180,E1 -19756.5,E2 -19756.5} C_VEL
LIN {X 0,Y 263.493,Z 371.092,A -85,B 0,C 180,E1 -19757.728,E2 -19757.728} C_VEL
LIN {X 0,Y 257.26,Z 357.967,A -85,B 0,C 180,E1 -19759.354,E2 -19759.354} C_VEL
LIN {X 0,Y 250.813,Z 345.963,A -85,B 0,C 180,E1 -19761.109,E2 -19761.109} C_VEL
LIN {X 0,Y 245.271,Z 336.971,A -85,B 0,C 180,E1 -19762.684,E2 -19762.684} C_VEL
LIN {X 0,Y 240.772,Z 330.364,A -85,B 0,C 180,E1 -19764.024,E2 -19764.024} C_VEL
LIN {X 0,Y 238.459,Z 327.041,A -85,B 0,C 180,E1 -19764.747,E2 -19764.747} C_VEL
LIN {X 0,Y 237.75,Z 326.058,A -85,B 0,C 180,E1 -19764.972,E2 -19764.972} C_VEL
LIN {X 0,Y 235.733,Z 323.758,A -85,B 0,C 180,E1 -19765.602,E2 -19765.602} C_VEL
LIN {X 0,Y 234.909,Z 321.223,A -85,B 0,C 180,E1 -19765.938,E2 -19765.938} C_VEL
LIN {X 0,Y 234.972,Z 321.208,A -85,B 0,C 180,E1 -19770.157,E2 -19770.157} C_VEL
LIN {X 0,Y 234.997,Z 321.205,A -85,B 0,C 180,E1 -19773.794,E2 -19773.794} C_VEL
LIN {X 0,Y 235.014,Z 321.211,A -85,B 0,C 180,E1 -19778.97,E2 -19778.97} C_VEL
LIN {X 0,Y 235.099,Z 321.198,A -85,B 0,C 180,E1 -19783.059,E2 -19783.059} C_VEL
LIN {X 0,Y 235.149,Z 321.195,A -85,B 0,C 180,E1 -19787.924,E2 -19787.924} C_VEL
LIN {X 0,Y 235.38,Z 321.151,A -85,B 0,C 180,E1 -19791.414,E2 -19791.414} C_VEL
LIN {X 0,Y 235.406,Z 321.162,A -85,B 0,C 180,E1 -19793.141,E2 -19793.141} C_VEL
LIN {X 0,Y 235.597,Z 321.137,A -85,B 0,C 180,E1 -19798.29,E2 -19798.29} C_VEL
LIN {X 0,Y 235.597,Z 321.12,A -85,B 0,C 180,E1 -19801.709,E2 -19801.709} C_VEL
LIN {X 0,Y 235.408,Z 321.145,A -85,B 0,C 180,E1 -19806.858,E2 -19806.858} C_VEL
LIN {X 0,Y 235.256,Z 321.164,A -85,B 0,C 180,E1 -19810.326,E2 -19810.326} C_VEL
LIN {X 0,Y 235.116,Z 321.184,A -85,B 0,C 180,E1 -19815.606,E2 -19815.606} C_VEL
LIN {X 0,Y 235.01,Z 321.209,A -85,B 0,C 180,E1 -19819.205,E2 -19819.205} C_VEL
LIN {X 0,Y 234.996,Z 321.198,A -85,B 0,C 180,E1 -19820.944,E2 -19820.944} C_VEL
LIN {X 0,Y 234.718,Z 321.238,A -85,B 0,C 180,E1 -19821.901,E2 -19821.901} C_VEL
LIN {X 0,Y 233.382,Z 321.415,A -85,B 0,C 180,E1 -19823.313,E2 -19823.313} C_VEL
LIN {X 0,Y 228.997,Z 321.956,A -85,B 0,C 180,E1 -19826.609,E2 -19826.609} C_VEL
LIN {X 0,Y 227.946,Z 322.091,A -85,B 0,C 180,E1 -19828.088,E2 -19828.088} C_VEL
LIN {X 0,Y 227.871,Z 322.089,A -85,B 0,C 180,E1 -19828.59,E2 -19828.59} C_VEL
LIN {X 0,Y 227.873,Z 322.098,A -85,B 0,C 180,E1 -19831.622,E2 -19831.622} C_VEL
LIN {X 0,Y 227.884,Z 322.099,A -85,B 0,C 180,E1 -19835.871,E2 -19835.871} C_VEL
LIN {X 0,Y 227.843,Z 322.176,A -85,B 0,C 180,E1 -19840.793,E2 -19840.793} C_VEL
LIN {X 0,Y 230.412,Z 330.406,A -85,B 0,C 180,E1 -19845.846,E2 -19845.846} C_VEL
LIN {X 0,Y 231.16,Z 332.757,A -85,B 0,C 180,E1 -19847.1,E2 -19847.1} C_VEL
LIN {X 0,Y 233.805,Z 337.275,A -85,B 0,C 180,E1 -19848.03,E2 -19848.03} C_VEL
LIN {X 0,Y 235.718,Z 340.42,A -85,B 0,C 180,E1 -19848.674,E2 -19848.674} C_VEL
LIN {X 0,Y 238.758,Z 345.376,A -85,B 0,C 180,E1 -19849.658,E2 -19849.658} C_VEL
LIN {X 0,Y 244.017,Z 354.766,A -85,B 0,C 180,E1 -19851.291,E2 -19851.291} C_VEL
LIN {X 0,Y 250.76,Z 368.304,A -85,B 0,C 180,E1 -19853.277,E2 -19853.277} C_VEL
LIN {X 0,Y 254.774,Z 377.442,A -85,B 0,C 180,E1 -19854.419,E2 -19854.419} C_VEL
LIN {X 0,Y 257.11,Z 392.776,A -85,B 0,C 180,E1 -19855.421,E2 -19855.421} C_VEL
LIN {X 0,Y 254.558,Z 443.4,A -85,B 0,C 180,E1 -19856.838,E2 -19856.838} C_VEL
LIN {X 0,Y 253.035,Z 456.961,A -85,B 0,C 180,E1 -19857.501,E2 -19857.501} C_VEL
LIN {X 0,Y 250.847,Z 469.761,A -85,B 0,C 180,E1 -19858.427,E2 -19858.427} C_VEL
LIN {X 0,Y 248.279,Z 481.447,A -85,B 0,C 180,E1 -19859.602,E2 -19859.602} C_VEL
LIN {X 0,Y 245.259,Z 492.744,A -85,B 0,C 180,E1 -19861.081,E2 -19861.081} C_VEL
LIN {X 0,Y 242.251,Z 502.947,A -85,B 0,C 180,E1 -19862.81,E2 -19862.81} C_VEL
LIN {X 0,Y 239.005,Z 512.153,A -85,B 0,C 180,E1 -19864.761,E2 -19864.761} C_VEL
LIN {X 0,Y 235.664,Z 521.113,A -85,B 0,C 180,E1 -19867.188,E2 -19867.188} C_VEL
LIN {X 0,Y 232.973,Z 528.353,A -85,B 0,C 180,E1 -19869.7,E2 -19869.7} C_VEL
LIN {X 0,Y 230.672,Z 534.183,A -85,B 0,C 180,E1 -19872.26,E2 -19872.26} C_VEL
LIN {X 0,Y 228.654,Z 538.801,A -85,B 0,C 180,E1 -19874.854,E2 -19874.854} C_VEL
LIN {X 0,Y 227.283,Z 542.341,A -85,B 0,C 180,E1 -19877.498,E2 -19877.498} C_VEL
LIN {X 0,Y 226.61,Z 544.16,A -85,B 0,C 180,E1 -19879.275,E2 -19879.275} C_VEL
LIN {X 0,Y 225.822,Z 546.549,A -85,B 0,C 180,E1 -19882.848,E2 -19882.848} C_VEL
LIN {X 0,Y 225.676,Z 547.279,A -85,B 0,C 180,E1 -19885.236,E2 -19885.236} C_VEL
LIN {X 0,Y 225.721,Z 547.192,A -85,B 0,C 180,E1 -19888.214,E2 -19888.214} C_VEL
LIN {X 0,Y 225.819,Z 546.604,A -85,B 0,C 180,E1 -19889.999,E2 -19889.999} C_VEL
LIN {X 0,Y 225.765,Z 545.613,A -85,B 0,C 180,E1 -19891.783,E2 -19891.783} C_VEL
LIN {X 0,Y 225.716,Z 542.874,A -85,B 0,C 180,E1 -19894.885,E2 -19894.885} C_VEL
LIN {X 0,Y 225.972,Z 538.644,A -85,B 0,C 180,E1 -19898.044,E2 -19898.044} C_VEL
LIN {X 0,Y 226.457,Z 533.827,A -85,B 0,C 180,E1 -19900.73,E2 -19900.73} C_VEL
LIN {X 0,Y 227.302,Z 527.72,A -85,B 0,C 180,E1 -19903.407,E2 -19903.407} C_VEL
LIN {X 0,Y 228.639,Z 520.11,A -85,B 0,C 180,E1 -19906.059,E2 -19906.059} C_VEL
LIN {X 0,Y 230.157,Z 511.708,A -85,B 0,C 180,E1 -19908.402,E2 -19908.402} C_VEL
LIN {X 0,Y 231.962,Z 501.719,A -85,B 0,C 180,E1 -19910.621,E2 -19910.621} C_VEL
LIN {X 0,Y 233.266,Z 493.498,A -85,B 0,C 180,E1 -19912.122,E2 -19912.122} C_VEL
LIN {X 0,Y 235.17,Z 482.018,A -85,B 0,C 180,E1 -19913.792,E2 -19913.792} C_VEL
LIN {X 0,Y 236.841,Z 470.052,A -85,B 0,C 180,E1 -19915.13,E2 -19915.13} C_VEL
LIN {X 0,Y 238.216,Z 457.535,A -85,B 0,C 180,E1 -19916.147,E2 -19916.147} C_VEL
LIN {X 0,Y 239.307,Z 443.573,A -85,B 0,C 180,E1 -19916.899,E2 -19916.899} C_VEL
LIN {X 0,Y 241.111,Z 386.927,A -85,B 0,C 180,E1 -19918.587,E2 -19918.587} C_VEL
LIN {X 0,Y 236.837,Z 351.393,A -85,B 0,C 180,E1 -19920.201,E2 -19920.201} C_VEL
LIN {X 0,Y 231.379,Z 336.868,A -85,B 0,C 180,E1 -19921.319,E2 -19921.319} C_VEL
LIN {X 0,Y 230.554,Z 334.447,A -85,B 0,C 180,E1 -19921.544,E2 -19921.544} C_VEL
LIN {X 0,Y 228.612,Z 325.199,A -85,B 0,C 180,E1 -19925.288,E2 -19925.288} C_VEL
LIN {X 0,Y 227.881,Z 322.097,A -85,B 0,C 180,E1 -19926.692,E2 -19926.692} C_VEL
LIN {X 0,Y 227.821,Z 322.106,A -85,B 0,C 180,E1 -19930.375,E2 -19930.375} C_VEL
LIN {X 0,Y 227.826,Z 322.105,A -85,B 0,C 180,E1 -19935.192,E2 -19935.192} C_VEL
LIN {X 0,Y 227.83,Z 322.1,A -85,B 0,C 180,E1 -19939.624,E2 -19939.624} C_VEL
LIN {X 0,Y 227.895,Z 322.095,A -85,B 0,C 180,E1 -19944.131,E2 -19944.131} C_VEL
LIN {X 0,Y 227.867,Z 322.097,A -85,B 0,C 180,E1 -19948.377,E2 -19948.377} C_VEL
LIN {X 0,Y 227.88,Z 322.096,A -85,B 0,C 180,E1 -19952.444,E2 -19952.444} C_VEL
LIN {X 0,Y 227.908,Z 322.092,A -85,B 0,C 180,E1 -19956.367,E2 -19956.367} C_VEL
LIN {X 0,Y 227.936,Z 322.086,A -85,B 0,C 180,E1 -19960.174,E2 -19960.174} C_VEL
LIN {X 0,Y 228.05,Z 322.065,A -85,B 0,C 180,E1 -19963.897,E2 -19963.897} C_VEL
LIN {X 0,Y 228.086,Z 322.074,A -85,B 0,C 180,E1 -19967.544,E2 -19967.544} C_VEL
LIN {X 0,Y 228.299,Z 322.04,A -85,B 0,C 180,E1 -19971.146,E2 -19971.146} C_VEL
LIN {X 0,Y 228.348,Z 322.024,A -85,B 0,C 180,E1 -19972.928,E2 -19972.928} C_VEL
LIN {X 0,Y 228.547,Z 322.013,A -85,B 0,C 180,E1 -19978.238,E2 -19978.238} C_VEL
LIN {X 0,Y 228.546,Z 322.012,A -85,B 0,C 180,E1 -19981.762,E2 -19981.762} C_VEL
LIN {X 0,Y 228.303,Z 322.025,A -85,B 0,C 180,E1 -19987.073,E2 -19987.073} C_VEL
LIN {X 0,Y 228.139,Z 322.064,A -85,B 0,C 180,E1 -19990.652,E2 -19990.652} C_VEL
LIN {X 0,Y 228.058,Z 322.073,A -85,B 0,C 180,E1 -19994.273,E2 -19994.273} C_VEL
LIN {X 0,Y 227.996,Z 322.084,A -85,B 0,C 180,E1 -19997.954,E2 -19997.954} C_VEL
LIN {X 0,Y 227.91,Z 322.091,A -85,B 0,C 180,E1 -20002.322,E2 -20002.322} C_VEL
LIN {X 0,Y 227.937,Z 322.088,A -85,B 0,C 180,E1 -20006.604,E2 -20006.604} C_VEL
LIN {X 0,Y 227.903,Z 322.095,A -85,B 0,C 180,E1 -20010.297,E2 -20010.297} C_VEL
LIN {X 0,Y 227.872,Z 322.092,A -85,B 0,C 180,E1 -20013.722,E2 -20013.722} C_VEL
LIN {X 0,Y 227.838,Z 322.101,A -85,B 0,C 180,E1 -20018.093,E2 -20018.093} C_VEL
LIN {X 0,Y 227.781,Z 322.11,A -85,B 0,C 180,E1 -20022.75,E2 -20022.75} C_VEL
LIN {X 0,Y 227.781,Z 322.11,A -85,B 0,C 180,E1 -20027.253,E2 -20027.253} C_VEL
LIN {X 0,Y 227.837,Z 322.102,A -85,B 0,C 180,E1 -20031.91,E2 -20031.91} C_VEL
LIN {X 0,Y 227.876,Z 322.098,A -85,B 0,C 180,E1 -20036.379,E2 -20036.379} C_VEL
LIN {X 0,Y 227.874,Z 322.096,A -85,B 0,C 180,E1 -20040.433,E2 -20040.433} C_VEL
LIN {X 0,Y 227.901,Z 322.096,A -85,B 0,C 180,E1 -20044.424,E2 -20044.424} C_VEL
LIN {X 0,Y 227.951,Z 322.085,A -85,B 0,C 180,E1 -20048.288,E2 -20048.288} C_VEL
LIN {X 0,Y 227.978,Z 322.086,A -85,B 0,C 180,E1 -20052.334,E2 -20052.334} C_VEL
LIN {X 0,Y 228.973,Z 324.886,A -85,B 0,C 180,E1 -20052.574,E2 -20052.574} C_VEL
LIN {X 0,Y 235.051,Z 337.46,A -85,B 0,C 180,E1 -20053.731,E2 -20053.731} C_VEL
LIN {X 0,Y 241.829,Z 356.608,A -85,B 0,C 180,E1 -20055.111,E2 -20055.111} C_VEL
LIN {X 0,Y 241.893,Z 362.039,A -85,B 0,C 180,E1 -20055.293,E2 -20055.293} C_VEL
LIN {X 0,Y 239.549,Z 426.803,A -85,B 0,C 180,E1 -20057.182,E2 -20057.182} C_VEL
LIN {X 0,Y 238.723,Z 439.958,A -85,B 0,C 180,E1 -20057.893,E2 -20057.893} C_VEL
LIN {X 0,Y 237.449,Z 452.689,A -85,B 0,C 180,E1 -20058.909,E2 -20058.909} C_VEL
LIN {X 0,Y 236.133,Z 463.969,A -85,B 0,C 180,E1 -20060.147,E2 -20060.147} C_VEL
LIN {X 0,Y 234.504,Z 475.658,A -85,B 0,C 180,E1 -20061.826,E2 -20061.826} C_VEL
LIN {X 0,Y 232.731,Z 486.104,A -85,B 0,C 180,E1 -20063.717,E2 -20063.717} C_VEL
LIN {X 0,Y 231.129,Z 494.695,A -85,B 0,C 180,E1 -20065.642,E2 -20065.642} C_VEL
LIN {X 0,Y 229.613,Z 502.609,A -85,B 0,C 180,E1 -20067.809,E2 -20067.809} C_VEL
LIN {X 0,Y 228.17,Z 510.326,A -85,B 0,C 180,E1 -20070.442,E2 -20070.442} C_VEL
LIN {X 0,Y 227.265,Z 515.606,A -85,B 0,C 180,E1 -20072.66,E2 -20072.66} C_VEL
LIN {X 0,Y 226.524,Z 520.713,A -85,B 0,C 180,E1 -20075.342,E2 -20075.342} C_VEL
LIN {X 0,Y 225.928,Z 524.692,A -85,B 0,C 180,E1 -20078.048,E2 -20078.048} C_VEL
LIN {X 0,Y 225.543,Z 527.63,A -85,B 0,C 180,E1 -20080.777,E2 -20080.777} C_VEL
LIN {X 0,Y 225.482,Z 529.017,A -85,B 0,C 180,E1 -20082.603,E2 -20082.603} C_VEL
LIN {X 0,Y 225.538,Z 530.231,A -85,B 0,C 180,E1 -20084.984,E2 -20084.984} C_VEL
LIN {X 0,Y 225.754,Z 530.726,A -85,B 0,C 180,E1 -20088.139,E2 -20088.139} C_VEL
LIN {X 0,Y 226.573,Z 529.922,A -85,B 0,C 180,E1 -20091.477,E2 -20091.477} C_VEL
LIN {X 0,Y 227.334,Z 528.636,A -85,B 0,C 180,E1 -20093.698,E2 -20093.698} C_VEL
LIN {X 0,Y 229.084,Z 525.263,A -85,B 0,C 180,E1 -20097.166,E2 -20097.166} C_VEL
LIN {X 0,Y 231.053,Z 520.995,A -85,B 0,C 180,E1 -20100.126,E2 -20100.126} C_VEL
LIN {X 0,Y 233.374,Z 515.734,A -85,B 0,C 180,E1 -20102.825,E2 -20102.825} C_VEL
LIN {X 0,Y 236.158,Z 508.999,A -85,B 0,C 180,E1 -20105.474,E2 -20105.474} C_VEL
LIN {X 0,Y 239.386,Z 500.535,A -85,B 0,C 180,E1 -20108.064,E2 -20108.064} C_VEL
LIN {X 0,Y 242.467,Z 491.792,A -85,B 0,C 180,E1 -20110.161,E2 -20110.161} C_VEL
LIN {X 0,Y 245.576,Z 481.832,A -85,B 0,C 180,E1 -20112.043,E2 -20112.043} C_VEL
LIN {X 0,Y 248.355,Z 471.386,A -85,B 0,C 180,E1 -20113.613,E2 -20113.613} C_VEL
LIN {X 0,Y 250.827,Z 460.075,A -85,B 0,C 180,E1 -20114.952,E2 -20114.952} C_VEL
LIN {X 0,Y 253.017,Z 447.517,A -85,B 0,C 180,E1 -20116.054,E2 -20116.054} C_VEL
LIN {X 0,Y 254.562,Z 434.592,A -85,B 0,C 180,E1 -20116.862,E2 -20116.862} C_VEL
LIN {X 0,Y 255.524,Z 421.701,A -85,B 0,C 180,E1 -20117.365,E2 -20117.365} C_VEL
LIN {X 0,Y 257.983,Z 373.434,A -85,B 0,C 180,E1 -20118.652,E2 -20118.652} C_VEL
LIN {X 0,Y 251.705,Z 360.361,A -85,B 0,C 180,E1 -20120.369,E2 -20120.369} C_VEL
LIN {X 0,Y 245.921,Z 349.653,A -85,B 0,C 180,E1 -20122.024,E2 -20122.024} C_VEL
LIN {X 0,Y 241.038,Z 341.551,A -85,B 0,C 180,E1 -20123.488,E2 -20123.488} C_VEL
LIN {X 0,Y 236.694,Z 335.317,A -85,B 0,C 180,E1 -20124.836,E2 -20124.836} C_VEL
LIN {X 0,Y 234.116,Z 331.585,A -85,B 0,C 180,E1 -20125.681,E2 -20125.681} C_VEL
LIN {X 0,Y 231.815,Z 328.567,A -85,B 0,C 180,E1 -20126.448,E2 -20126.448} C_VEL
LIN {X 0,Y 230.896,Z 327.026,A -85,B 0,C 180,E1 -20126.778,E2 -20126.778} C_VEL
LIN {X 0,Y 228.811,Z 324.76,A -85,B 0,C 180,E1 -20127.485,E2 -20127.485} C_VEL
LIN {X 0,Y 227.894,Z 322.095,A -85,B 0,C 180,E1 -20127.926,E2 -20127.926} C_VEL
LIN {X 0,Y 227.922,Z 322.087,A -85,B 0,C 180,E1 -20130.438,E2 -20130.438} C_VEL
LIN {X 0,Y 227.932,Z 322.089,A -85,B 0,C 180,E1 -20134.426,E2 -20134.426} C_VEL
LIN {X 0,Y 227.965,Z 322.084,A -85,B 0,C 180,E1 -20138.287,E2 -20138.287} C_VEL
LIN {X 0,Y 228.038,Z 322.077,A -85,B 0,C 180,E1 -20142.826,E2 -20142.826} C_VEL
LIN {X 0,Y 228.097,Z 322.07,A -85,B 0,C 180,E1 -20147.544,E2 -20147.544} C_VEL
LIN {X 0,Y 228.309,Z 322.03,A -85,B 0,C 180,E1 -20151.146,E2 -20151.146} C_VEL
LIN {X 0,Y 228.357,Z 322.04,A -85,B 0,C 180,E1 -20152.929,E2 -20152.929} C_VEL
LIN {X 0,Y 228.556,Z 322.014,A -85,B 0,C 180,E1 -20158.238,E2 -20158.238} C_VEL
LIN {X 0,Y 228.556,Z 321.997,A -85,B 0,C 180,E1 -20161.762,E2 -20161.762} C_VEL
LIN {X 0,Y 228.36,Z 322.023,A -85,B 0,C 180,E1 -20167.071,E2 -20167.071} C_VEL
LIN {X 0,Y 228.17,Z 322.045,A -85,B 0,C 180,E1 -20170.65,E2 -20170.65} C_VEL
LIN {X 0,Y 228.068,Z 322.073,A -85,B 0,C 180,E1 -20174.272,E2 -20174.272} C_VEL
LIN {X 0,Y 228.006,Z 322.079,A -85,B 0,C 180,E1 -20177.953,E2 -20177.953} C_VEL
LIN {X 0,Y 227.919,Z 322.086,A -85,B 0,C 180,E1 -20182.321,E2 -20182.321} C_VEL
LIN {X 0,Y 227.946,Z 322.08,A -85,B 0,C 180,E1 -20186.602,E2 -20186.602} C_VEL
LIN {X 0,Y 227.871,Z 322.089,A -85,B 0,C 180,E1 -20188.59,E2 -20188.59} C_VEL
LIN {X 0,Y 227.214,Z 322.17,A -85,B 0,C 180,E1 -20190.065,E2 -20190.065} C_VEL
LIN {X 0,Y 224.321,Z 322.539,A -85,B 0,C 180,E1 -20192.471,E2 -20192.471} C_VEL
LIN {X 0,Y 221.869,Z 322.839,A -85,B 0,C 180,E1 -20194.435,E2 -20194.435} C_VEL
LIN {X 0,Y 220.848,Z 322.975,A -85,B 0,C 180,E1 -20195.961,E2 -20195.961} C_VEL
LIN {X 0,Y 220.782,Z 322.971,A -85,B 0,C 180,E1 -20196.479,E2 -20196.479} C_VEL
LIN {X 0,Y 220.815,Z 323.13,A -85,B 0,C 180,E1 -20198.946,E2 -20198.946} C_VEL
LIN {X 0,Y 223.119,Z 330.531,A -85,B 0,C 180,E1 -20203.866,E2 -20203.866} C_VEL
LIN {X 0,Y 223.748,Z 332.272,A -85,B 0,C 180,E1 -20204.89,E2 -20204.89} C_VEL
LIN {X 0,Y 226.488,Z 336.795,A -85,B 0,C 180,E1 -20205.948,E2 -20205.948} C_VEL
LIN {X 0,Y 227.997,Z 339.04,A -85,B 0,C 180,E1 -20206.498,E2 -20206.498} C_VEL
LIN {X 0,Y 234.325,Z 349.404,A -85,B 0,C 180,E1 -20208.712,E2 -20208.712} C_VEL
LIN {X 0,Y 240.506,Z 360.759,A -85,B 0,C 180,E1 -20210.726,E2 -20210.726} C_VEL
LIN {X 0,Y 246.937,Z 374.164,A -85,B 0,C 180,E1 -20212.706,E2 -20212.706} C_VEL
LIN {X 0,Y 249.666,Z 380.523,A -85,B 0,C 180,E1 -20213.52,E2 -20213.52} C_VEL
LIN {X 0,Y 251.652,Z 393.969,A -85,B 0,C 180,E1 -20214.425,E2 -20214.425} C_VEL
LIN {X 0,Y 249.035,Z 443.181,A -85,B 0,C 180,E1 -20215.821,E2 -20215.821} C_VEL
LIN {X 0,Y 247.433,Z 456.734,A -85,B 0,C 180,E1 -20216.488,E2 -20216.488} C_VEL
LIN {X 0,Y 245.296,Z 469.007,A -85,B 0,C 180,E1 -20217.384,E2 -20217.384} C_VEL
LIN {X 0,Y 242.617,Z 480.805,A -85,B 0,C 180,E1 -20218.572,E2 -20218.572} C_VEL
LIN {X 0,Y 239.492,Z 492.162,A -85,B 0,C 180,E1 -20220.074,E2 -20220.074} C_VEL
LIN {X 0,Y 236.292,Z 502.423,A -85,B 0,C 180,E1 -20221.824,E2 -20221.824} C_VEL
LIN {X 0,Y 233.244,Z 510.841,A -85,B 0,C 180,E1 -20223.611,E2 -20223.611} C_VEL
LIN {X 0,Y 229.668,Z 519.993,A -85,B 0,C 180,E1 -20226.079,E2 -20226.079} C_VEL
LIN {X 0,Y 226.899,Z 527.035,A -85,B 0,C 180,E1 -20228.51,E2 -20228.51} C_VEL
LIN {X 0,Y 224.65,Z 532.432,A -85,B 0,C 180,E1 -20230.822,E2 -20230.822} C_VEL
LIN {X 0,Y 222.426,Z 537.362,A -85,B 0,C 180,E1 -20233.477,E2 -20233.477} C_VEL
LIN {X 0,Y 220.724,Z 541.192,A -85,B 0,C 180,E1 -20236.183,E2 -20236.183} C_VEL
LIN {X 0,Y 219.62,Z 544.026,A -85,B 0,C 180,E1 -20238.929,E2 -20238.929} C_VEL
LIN {X 0,Y 218.761,Z 546.356,A -85,B 0,C 180,E1 -20242.616,E2 -20242.616} C_VEL
LIN {X 0,Y 218.57,Z 547.062,A -85,B 0,C 180,E1 -20245.409,E2 -20245.409} C_VEL
LIN {X 0,Y 218.633,Z 546.883,A -85,B 0,C 180,E1 -20248.157,E2 -20248.157} C_VEL
LIN {X 0,Y 218.751,Z 546.267,A -85,B 0,C 180,E1 -20249.999,E2 -20249.999} C_VEL
LIN {X 0,Y 218.676,Z 545.246,A -85,B 0,C 180,E1 -20251.84,E2 -20251.84} C_VEL
LIN {X 0,Y 218.616,Z 542.747,A -85,B 0,C 180,E1 -20254.741,E2 -20254.741} C_VEL
LIN {X 0,Y 218.828,Z 539.496,A -85,B 0,C 180,E1 -20257.38,E2 -20257.38} C_VEL
LIN {X 0,Y 219.234,Z 535.006,A -85,B 0,C 180,E1 -20260.154,E2 -20260.154} C_VEL
LIN {X 0,Y 220.159,Z 528.173,A -85,B 0,C 180,E1 -20263.38,E2 -20263.38} C_VEL
LIN {X 0,Y 221.544,Z 520.721,A -85,B 0,C 180,E1 -20266.114,E2 -20266.114} C_VEL
LIN {X 0,Y 223.183,Z 511.794,A -85,B 0,C 180,E1 -20268.729,E2 -20268.729} C_VEL
LIN {X 0,Y 225.08,Z 501.745,A -85,B 0,C 180,E1 -20271.042,E2 -20271.042} C_VEL
LIN {X 0,Y 226.432,Z 493.585,A -85,B 0,C 180,E1 -20272.586,E2 -20272.586} C_VEL
LIN {X 0,Y 228.388,Z 482.181,A -85,B 0,C 180,E1 -20274.302,E2 -20274.302} C_VEL
LIN {X 0,Y 230.112,Z 470.334,A -85,B 0,C 180,E1 -20275.676,E2 -20275.676} C_VEL
LIN {X 0,Y 231.609,Z 457.326,A -85,B 0,C 180,E1 -20276.769,E2 -20276.769} C_VEL
LIN {X 0,Y 232.705,Z 443.853,A -85,B 0,C 180,E1 -20277.519,E2 -20277.519} C_VEL
LIN {X 0,Y 234.585,Z 387.698,A -85,B 0,C 180,E1 -20279.243,E2 -20279.243} C_VEL
LIN {X 0,Y 230.557,Z 353.395,A -85,B 0,C 180,E1 -20280.853,E2 -20280.853} C_VEL
LIN {X 0,Y 224.254,Z 336.858,A -85,B 0,C 180,E1 -20282.203,E2 -20282.203} C_VEL
LIN {X 0,Y 223.3,Z 334.167,A -85,B 0,C 180,E1 -20282.462,E2 -20282.462} C_VEL
LIN {X 0,Y 221.513,Z 325.923,A -85,B 0,C 180,E1 -20285.939,E2 -20285.939} C_VEL
LIN {X 0,Y 220.804,Z 322.978,A -85,B 0,C 180,E1 -20287.276,E2 -20287.276} C_VEL
LIN {X 0,Y 220.79,Z 322.981,A -85,B 0,C 180,E1 -20290.186,E2 -20290.186} C_VEL
LIN {X 0,Y 220.766,Z 322.986,A -85,B 0,C 180,E1 -20294.453,E2 -20294.453} C_VEL
LIN {X 0,Y 220.771,Z 322.985,A -85,B 0,C 180,E1 -20298.048,E2 -20298.048} C_VEL
LIN {X 0,Y 220.827,Z 322.979,A -85,B 0,C 180,E1 -20302.793,E2 -20302.793} C_VEL
LIN {X 0,Y 220.819,Z 322.975,A -85,B 0,C 180,E1 -20307.244,E2 -20307.244} C_VEL
LIN {X 0,Y 220.831,Z 322.974,A -85,B 0,C 180,E1 -20311.486,E2 -20311.486} C_VEL
LIN {X 0,Y 220.861,Z 322.971,A -85,B 0,C 180,E1 -20315.564,E2 -20315.564} C_VEL
LIN {X 0,Y 220.886,Z 322.966,A -85,B 0,C 180,E1 -20319.513,E2 -20319.513} C_VEL
LIN {X 0,Y 221.009,Z 322.937,A -85,B 0,C 180,E1 -20323.37,E2 -20323.37} C_VEL
LIN {X 0,Y 221.105,Z 322.943,A -85,B 0,C 180,E1 -20329.006,E2 -20329.006} C_VEL
LIN {X 0,Y 221.283,Z 322.905,A -85,B 0,C 180,E1 -20332.701,E2 -20332.701} C_VEL
LIN {X 0,Y 221.505,Z 322.89,A -85,B 0,C 180,E1 -20338.182,E2 -20338.182} C_VEL
LIN {X 0,Y 221.504,Z 322.889,A -85,B 0,C 180,E1 -20341.818,E2 -20341.818} C_VEL
LIN {X 0,Y 221.24,Z 322.905,A -85,B 0,C 180,E1 -20347.3,E2 -20347.3} C_VEL
LIN {X 0,Y 221.06,Z 322.945,A -85,B 0,C 180,E1 -20350.997,E2 -20350.997} C_VEL
LIN {X 0,Y 220.989,Z 322.951,A -85,B 0,C 180,E1 -20354.739,E2 -20354.739} C_VEL
LIN {X 0,Y 220.914,Z 322.967,A -85,B 0,C 180,E1 -20358.55,E2 -20358.55} C_VEL
LIN {X 0,Y 220.879,Z 322.969,A -85,B 0,C 180,E1 -20362.676,E2 -20362.676} C_VEL
LIN {X 0,Y 220.88,Z 322.965,A -85,B 0,C 180,E1 -20367.017,E2 -20367.017} C_VEL
LIN {X 0,Y 220.858,Z 322.973,A -85,B 0,C 180,E1 -20370.78,E2 -20370.78} C_VEL
LIN {X 0,Y 220.796,Z 322.98,A -85,B 0,C 180,E1 -20374.956,E2 -20374.956} C_VEL
LIN {X 0,Y 220.804,Z 322.977,A -85,B 0,C 180,E1 -20377.279,E2 -20377.279} C_VEL
LIN {X 0,Y 220.743,Z 322.985,A -85,B 0,C 180,E1 -20381.959,E2 -20381.959} C_VEL
LIN {X 0,Y 220.748,Z 322.985,A -85,B 0,C 180,E1 -20385.542,E2 -20385.542} C_VEL
LIN {X 0,Y 220.777,Z 322.982,A -85,B 0,C 180,E1 -20390.459,E2 -20390.459} C_VEL
LIN {X 0,Y 220.822,Z 322.977,A -85,B 0,C 180,E1 -20392.795,E2 -20392.795} C_VEL
LIN {X 0,Y 220.81,Z 322.978,A -85,B 0,C 180,E1 -20397.245,E2 -20397.245} C_VEL
LIN {X 0,Y 220.802,Z 322.982,A -85,B 0,C 180,E1 -20401.484,E2 -20401.484} C_VEL
LIN {X 0,Y 220.846,Z 322.975,A -85,B 0,C 180,E1 -20405.564,E2 -20405.564} C_VEL
LIN {X 0,Y 220.878,Z 322.968,A -85,B 0,C 180,E1 -20409.514,E2 -20409.514} C_VEL
LIN {X 0,Y 220.891,Z 322.967,A -85,B 0,C 180,E1 -20411.45,E2 -20411.45} C_VEL
LIN {X 0,Y 221.857,Z 325.741,A -85,B 0,C 180,E1 -20411.689,E2 -20411.689} C_VEL
LIN {X 0,Y 228.618,Z 339.309,A -85,B 0,C 180,E1 -20413.029,E2 -20413.029} C_VEL
LIN {X 0,Y 235.441,Z 358.406,A -85,B 0,C 180,E1 -20414.476,E2 -20414.476} C_VEL
LIN {X 0,Y 232.995,Z 427.025,A -85,B 0,C 180,E1 -20416.538,E2 -20416.538} C_VEL
LIN {X 0,Y 232.117,Z 440.204,A -85,B 0,C 180,E1 -20417.265,E2 -20417.265} C_VEL
LIN {X 0,Y 230.734,Z 453.497,A -85,B 0,C 180,E1 -20418.36,E2 -20418.36} C_VEL
LIN {X 0,Y 229.376,Z 464.619,A -85,B 0,C 180,E1 -20419.631,E2 -20419.631} C_VEL
LIN {X 0,Y 227.656,Z 476.47,A -85,B 0,C 180,E1 -20421.396,E2 -20421.396} C_VEL
LIN {X 0,Y 225.855,Z 486.628,A -85,B 0,C 180,E1 -20423.3,E2 -20423.3} C_VEL
LIN {X 0,Y 224.017,Z 496.032,A -85,B 0,C 180,E1 -20425.503,E2 -20425.503} C_VEL
LIN {X 0,Y 222.228,Z 505.103,A -85,B 0,C 180,E1 -20428.189,E2 -20428.189} C_VEL
LIN {X 0,Y 220.843,Z 512.412,A -85,B 0,C 180,E1 -20430.913,E2 -20430.913} C_VEL
LIN {X 0,Y 219.814,Z 518.262,A -85,B 0,C 180,E1 -20433.668,E2 -20433.668} C_VEL
LIN {X 0,Y 219.194,Z 522.652,A -85,B 0,C 180,E1 -20436.303,E2 -20436.303} C_VEL
LIN {X 0,Y 218.624,Z 526.377,A -85,B 0,C 180,E1 -20439.251,E2 -20439.251} C_VEL
LIN {X 0,Y 218.416,Z 528.129,A -85,B 0,C 180,E1 -20441.133,E2 -20441.133} C_VEL
LIN {X 0,Y 218.388,Z 529.465,A -85,B 0,C 180,E1 -20443.02,E2 -20443.02} C_VEL
LIN {X 0,Y 218.462,Z 530.497,A -85,B 0,C 180,E1 -20445.178,E2 -20445.178} C_VEL
LIN {X 0,Y 218.758,Z 530.972,A -85,B 0,C 180,E1 -20448.741,E2 -20448.741} C_VEL
LIN {X 0,Y 219.565,Z 530.212,A -85,B 0,C 180,E1 -20451.835,E2 -20451.835} C_VEL
LIN {X 0,Y 220.543,Z 528.673,A -85,B 0,C 180,E1 -20454.474,E2 -20454.474} C_VEL
LIN {X 0,Y 222.23,Z 525.604,A -85,B 0,C 180,E1 -20457.687,E2 -20457.687} C_VEL
LIN {X 0,Y 224.634,Z 520.777,A -85,B 0,C 180,E1 -20461.081,E2 -20461.081} C_VEL
LIN {X 0,Y 227.136,Z 515.354,A -85,B 0,C 180,E1 -20463.846,E2 -20463.846} C_VEL
LIN {X 0,Y 230.131,Z 508.474,A -85,B 0,C 180,E1 -20466.55,E2 -20466.55} C_VEL
LIN {X 0,Y 233.076,Z 501.086,A -85,B 0,C 180,E1 -20468.844,E2 -20468.844} C_VEL
LIN {X 0,Y 236.158,Z 492.789,A -85,B 0,C 180,E1 -20470.899,E2 -20470.899} C_VEL
LIN {X 0,Y 239.537,Z 482.539,A -85,B 0,C 180,E1 -20472.904,E2 -20472.904} C_VEL
LIN {X 0,Y 242.646,Z 471.327,A -85,B 0,C 180,E1 -20474.619,E2 -20474.619} C_VEL
LIN {X 0,Y 245.23,Z 459.954,A -85,B 0,C 180,E1 -20475.974,E2 -20475.974} C_VEL
LIN {X 0,Y 247.454,Z 447.45,A -85,B 0,C 180,E1 -20477.078,E2 -20477.078} C_VEL
LIN {X 0,Y 249.092,Z 434.317,A -85,B 0,C 180,E1 -20477.897,E2 -20477.897} C_VEL
LIN {X 0,Y 250.08,Z 420.79,A -85,B 0,C 180,E1 -20478.415,E2 -20478.415} C_VEL
LIN {X 0,Y 252.506,Z 375.824,A -85,B 0,C 180,E1 -20479.623,E2 -20479.623} C_VEL
LIN {X 0,Y 245.696,Z 361.707,A -85,B 0,C 180,E1 -20481.592,E2 -20481.592} C_VEL
LIN {X 0,Y 239.775,Z 350.976,A -85,B 0,C 180,E1 -20483.395,E2 -20483.395} C_VEL
LIN {X 0,Y 235.39,Z 344.052,A -85,B 0,C 180,E1 -20484.787,E2 -20484.787} C_VEL
LIN {X 0,Y 230.178,Z 336.633,A -85,B 0,C 180,E1 -20486.53,E2 -20486.53} C_VEL
LIN {X 0,Y 226.985,Z 332.237,A -85,B 0,C 180,E1 -20487.662,E2 -20487.662} C_VEL
LIN {X 0,Y 224.778,Z 329.118,A -85,B 0,C 180,E1 -20488.484,E2 -20488.484} C_VEL
LIN {X 0,Y 223.918,Z 327.959,A -85,B 0,C 180,E1 -20488.81,E2 -20488.81} C_VEL
LIN {X 0,Y 221.915,Z 325.907,A -85,B 0,C 180,E1 -20489.554,E2 -20489.554} C_VEL
LIN {X 0,Y 220.956,Z 323.423,A -85,B 0,C 180,E1 -20490.002,E2 -20490.002} C_VEL
LIN {X 0,Y 220.869,Z 322.965,A -85,B 0,C 180,E1 -20490.12,E2 -20490.12} C_VEL
LIN {X 0,Y 220.899,Z 322.96,A -85,B 0,C 180,E1 -20493.55,E2 -20493.55} C_VEL
LIN {X 0,Y 220.881,Z 322.96,A -85,B 0,C 180,E1 -20497.554,E2 -20497.554} C_VEL
LIN {X 0,Y 220.988,Z 322.952,A -85,B 0,C 180,E1 -20502.571,E2 -20502.571} C_VEL
LIN {X 0,Y 221.029,Z 322.946,A -85,B 0,C 180,E1 -20507.139,E2 -20507.139} C_VEL
LIN {X 0,Y 221.239,Z 322.909,A -85,B 0,C 180,E1 -20510.861,E2 -20510.861} C_VEL
LIN {X 0,Y 221.308,Z 322.918,A -85,B 0,C 180,E1 -20512.702,E2 -20512.702} C_VEL
LIN {X 0,Y 221.514,Z 322.892,A -85,B 0,C 180,E1 -20518.182,E2 -20518.182} C_VEL
LIN {X 0,Y 221.514,Z 322.874,A -85,B 0,C 180,E1 -20521.818,E2 -20521.818} C_VEL
LIN {X 0,Y 221.313,Z 322.903,A -85,B 0,C 180,E1 -20527.298,E2 -20527.298} C_VEL
LIN {X 0,Y 221.114,Z 322.922,A -85,B 0,C 180,E1 -20530.994,E2 -20530.994} C_VEL
LIN {X 0,Y 221.019,Z 322.937,A -85,B 0,C 180,E1 -20536.63,E2 -20536.63} C_VEL
LIN {X 0,Y 220.887,Z 322.957,A -85,B 0,C 180,E1 -20540.487,E2 -20540.487} C_VEL
LIN {X 0,Y 220.865,Z 322.966,A -85,B 0,C 180,E1 -20544.435,E2 -20544.435} C_VEL
LIN {X 0,Y 220.837,Z 322.972,A -85,B 0,C 180,E1 -20548.567,E2 -20548.567} C_VEL
LIN {X 0,Y 220.821,Z 322.972,A -85,B 0,C 180,E1 -20552.755,E2 -20552.755} C_VEL
LIN {X 0,Y 220.782,Z 322.971,A -85,B 0,C 180,E1 -20556.479,E2 -20556.479} C_VEL
LIN {X 0,Y 220.267,Z 323.469,A -85,B 0,C 180,E1 -20557.487,E2 -20557.487} C_VEL
LIN {X 0,Y 218.079,Z 325.75,A -85,B 0,C 180,E1 -20559.034,E2 -20559.034} C_VEL
LIN {X 0,Y 216.05,Z 328.793,A -85,B 0,C 180,E1 -20560.569,E2 -20560.569} C_VEL
LIN {X 0,Y 215.847,Z 330.477,A -85,B 0,C 180,E1 -20561.549,E2 -20561.549} C_VEL
LIN {X 0,Y 216.341,Z 331.975,A -85,B 0,C 180,E1 -20562.404,E2 -20562.404} C_VEL
LIN {X 0,Y 219.099,Z 336.342,A -85,B 0,C 180,E1 -20563.597,E2 -20563.597} C_VEL
LIN {X 0,Y 220.688,Z 338.44,A -85,B 0,C 180,E1 -20564.232,E2 -20564.232} C_VEL
LIN {X 0,Y 223.647,Z 342.978,A -85,B 0,C 180,E1 -20565.395,E2 -20565.395} C_VEL
LIN {X 0,Y 230.307,Z 354.124,A -85,B 0,C 180,E1 -20567.855,E2 -20567.855} C_VEL
LIN {X 0,Y 236.696,Z 366.106,A -85,B 0,C 180,E1 -20570.038,E2 -20570.038} C_VEL
LIN {X 0,Y 242.966,Z 379.651,A -85,B 0,C 180,E1 -20572.061,E2 -20572.061} C_VEL
LIN {X 0,Y 244.676,Z 384.017,A -85,B 0,C 180,E1 -20572.611,E2 -20572.611} C_VEL
LIN {X 0,Y 246.261,Z 395.098,A -85,B 0,C 180,E1 -20573.381,E2 -20573.381} C_VEL
LIN {X 0,Y 243.577,Z 442.972,A -85,B 0,C 180,E1 -20574.755,E2 -20574.755} C_VEL
LIN {X 0,Y 241.94,Z 456.496,A -85,B 0,C 180,E1 -20575.433,E2 -20575.433} C_VEL
LIN {X 0,Y 239.613,Z 469.267,A -85,B 0,C 180,E1 -20576.384,E2 -20576.384} C_VEL
LIN {X 0,Y 236.636,Z 481.731,A -85,B 0,C 180,E1 -20577.683,E2 -20577.683} C_VEL
LIN {X 0,Y 233.41,Z 492.871,A -85,B 0,C 180,E1 -20579.21,E2 -20579.21} C_VEL
LIN {X 0,Y 230.439,Z 501.903,A -85,B 0,C 180,E1 -20580.792,E2 -20580.792} C_VEL
LIN {X 0,Y 226.929,Z 511.217,A -85,B 0,C 180,E1 -20582.818,E2 -20582.818} C_VEL
LIN {X 0,Y 223.209,Z 520.24,A -85,B 0,C 180,E1 -20585.342,E2 -20585.342} C_VEL
LIN {X 0,Y 220.145,Z 527.579,A -85,B 0,C 180,E1 -20587.988,E2 -20587.988} C_VEL
LIN {X 0,Y 217.132,Z 534.267,A -85,B 0,C 180,E1 -20591.114,E2 -20591.114} C_VEL
LIN {X 0,Y 214.953,Z 538.744,A -85,B 0,C 180,E1 -20593.863,E2 -20593.863} C_VEL
LIN {X 0,Y 213.353,Z 542.17,A -85,B 0,C 180,E1 -20596.667,E2 -20596.667} C_VEL
LIN {X 0,Y 212.069,Z 545.22,A -85,B 0,C 180,E1 -20600.461,E2 -20600.461} C_VEL
LIN {X 0,Y 211.507,Z 546.707,A -85,B 0,C 180,E1 -20604.278,E2 -20604.278} C_VEL
LIN {X 0,Y 211.486,Z 546.832,A -85,B 0,C 180,E1 -20606.188,E2 -20606.188} C_VEL
LIN {X 0,Y 211.548,Z 546.574,A -85,B 0,C 180,E1 -20608.095,E2 -20608.095} C_VEL
LIN {X 0,Y 211.684,Z 545.93,A -85,B 0,C 180,E1 -20609.999,E2 -20609.999} C_VEL
LIN {X 0,Y 211.589,Z 544.87,A -85,B 0,C 180,E1 -20611.902,E2 -20611.902} C_VEL
LIN {X 0,Y 211.535,Z 542.559,A -85,B 0,C 180,E1 -20614.644,E2 -20614.644} C_VEL
LIN {X 0,Y 211.744,Z 539,A -85,B 0,C 180,E1 -20617.628,E2 -20617.628} C_VEL
LIN {X 0,Y 212.189,Z 534.441,A -85,B 0,C 180,E1 -20620.494,E2 -20620.494} C_VEL
LIN {X 0,Y 213.22,Z 527.495,A -85,B 0,C 180,E1 -20623.824,E2 -20623.824} C_VEL
LIN {X 0,Y 214.649,Z 519.951,A -85,B 0,C 180,E1 -20626.646,E2 -20626.646} C_VEL
LIN {X 0,Y 216.183,Z 512.24,A -85,B 0,C 180,E1 -20628.97,E2 -20628.97} C_VEL
LIN {X 0,Y 218.011,Z 502.855,A -85,B 0,C 180,E1 -20631.262,E2 -20631.262} C_VEL
LIN {X 0,Y 219.613,Z 493.671,A -85,B 0,C 180,E1 -20633.079,E2 -20633.079} C_VEL
LIN {X 0,Y 221.626,Z 482.344,A -85,B 0,C 180,E1 -20634.844,E2 -20634.844} C_VEL
LIN {X 0,Y 223.405,Z 470.607,A -85,B 0,C 180,E1 -20636.254,E2 -20636.254} C_VEL
LIN {X 0,Y 224.921,Z 457.869,A -85,B 0,C 180,E1 -20637.379,E2 -20637.379} C_VEL
LIN {X 0,Y 226.121,Z 444.401,A -85,B 0,C 180,E1 -20638.162,E2 -20638.162} C_VEL
LIN {X 0,Y 227.221,Z 416.223,A -85,B 0,C 180,E1 -20639.083,E2 -20639.083} C_VEL
LIN {X 0,Y 228.002,Z 387.931,A -85,B 0,C 180,E1 -20639.966,E2 -20639.966} C_VEL
LIN {X 0,Y 224.377,Z 355.992,A -85,B 0,C 180,E1 -20641.509,E2 -20641.509} C_VEL
LIN {X 0,Y 218.843,Z 341.02,A -85,B 0,C 180,E1 -20642.759,E2 -20642.759} C_VEL
LIN {X 0,Y 216.02,Z 333.859,A -85,B 0,C 180,E1 -20643.456,E2 -20643.456} C_VEL
LIN {X 0,Y 214.017,Z 325.044,A -85,B 0,C 180,E1 -20647.365,E2 -20647.365} C_VEL
LIN {X 0,Y 213.732,Z 323.858,A -85,B 0,C 180,E1 -20647.965,E2 -20647.965} C_VEL
LIN {X 0,Y 213.707,Z 323.862,A -85,B 0,C 180,E1 -20651.124,E2 -20651.124} C_VEL
LIN {X 0,Y 213.699,Z 323.864,A -85,B 0,C 180,E1 -20653.678,E2 -20653.678} C_VEL
LIN {X 0,Y 213.702,Z 323.866,A -85,B 0,C 180,E1 -20656.342,E2 -20656.342} C_VEL
LIN {X 0,Y 213.731,Z 323.859,A -85,B 0,C 180,E1 -20661.335,E2 -20661.335} C_VEL
LIN {X 0,Y 213.764,Z 323.855,A -85,B 0,C 180,E1 -20666.019,E2 -20666.019} C_VEL
LIN {X 0,Y 213.775,Z 323.855,A -85,B 0,C 180,E1 -20670.453,E2 -20670.453} C_VEL
LIN {X 0,Y 213.796,Z 323.853,A -85,B 0,C 180,E1 -20674.701,E2 -20674.701} C_VEL
LIN {X 0,Y 213.807,Z 323.853,A -85,B 0,C 180,E1 -20678.803,E2 -20678.803} C_VEL
LIN {X 0,Y 213.937,Z 323.816,A -85,B 0,C 180,E1 -20682.803,E2 -20682.803} C_VEL
LIN {X 0,Y 213.972,Z 323.828,A -85,B 0,C 180,E1 -20686.708,E2 -20686.708} C_VEL
LIN {X 0,Y 214.161,Z 323.802,A -85,B 0,C 180,E1 -20690.556,E2 -20690.556} C_VEL
LIN {X 0,Y 214.221,Z 323.785,A -85,B 0,C 180,E1 -20692.459,E2 -20692.459} C_VEL
LIN {X 0,Y 214.438,Z 323.771,A -85,B 0,C 180,E1 -20698.122,E2 -20698.122} C_VEL
LIN {X 0,Y 214.543,Z 323.759,A -85,B 0,C 180,E1 -20700,E2 -20700} C_VEL
LIN {X 0,Y 214.437,Z 323.768,A -85,B 0,C 180,E1 -20701.878,E2 -20701.878} C_VEL
LIN {X 0,Y 214.181,Z 323.784,A -85,B 0,C 180,E1 -20707.542,E2 -20707.542} C_VEL
LIN {X 0,Y 213.992,Z 323.826,A -85,B 0,C 180,E1 -20711.365,E2 -20711.365} C_VEL
LIN {X 0,Y 213.926,Z 323.83,A -85,B 0,C 180,E1 -20715.238,E2 -20715.238} C_VEL
LIN {X 0,Y 213.83,Z 323.848,A -85,B 0,C 180,E1 -20719.188,E2 -20719.188} C_VEL
LIN {X 0,Y 213.805,Z 323.849,A -85,B 0,C 180,E1 -20723.232,E2 -20723.232} C_VEL
LIN {X 0,Y 213.823,Z 323.843,A -85,B 0,C 180,E1 -20727.451,E2 -20727.451} C_VEL
LIN {X 0,Y 213.772,Z 323.853,A -85,B 0,C 180,E1 -20731.737,E2 -20731.737} C_VEL
LIN {X 0,Y 213.739,Z 323.859,A -85,B 0,C 180,E1 -20736.29,E2 -20736.29} C_VEL
LIN {X 0,Y 213.693,Z 323.865,A -85,B 0,C 180,E1 -20741.13,E2 -20741.13} C_VEL
LIN {X 0,Y 213.696,Z 323.859,A -85,B 0,C 180,E1 -20743.681,E2 -20743.681} C_VEL
LIN {X 0,Y 213.697,Z 323.864,A -85,B 0,C 180,E1 -20746.347,E2 -20746.347} C_VEL
LIN {X 0,Y 213.701,Z 323.865,A -85,B 0,C 180,E1 -20751.331,E2 -20751.331} C_VEL
LIN {X 0,Y 213.751,Z 323.857,A -85,B 0,C 180,E1 -20756.019,E2 -20756.019} C_VEL
LIN {X 0,Y 213.748,Z 323.856,A -85,B 0,C 180,E1 -20760.451,E2 -20760.451} C_VEL
LIN {X 0,Y 213.78,Z 323.855,A -85,B 0,C 180,E1 -20764.701,E2 -20764.701} C_VEL
LIN {X 0,Y 213.799,Z 323.847,A -85,B 0,C 180,E1 -20768.804,E2 -20768.804} C_VEL
LIN {X 0,Y 213.831,Z 323.85,A -85,B 0,C 180,E1 -20770.476,E2 -20770.476} C_VEL
LIN {X 0,Y 214.792,Z 326.635,A -85,B 0,C 180,E1 -20770.748,E2 -20770.748} C_VEL
LIN {X 0,Y 222.034,Z 340.967,A -85,B 0,C 180,E1 -20772.261,E2 -20772.261} C_VEL
LIN {X 0,Y 226.681,Z 353.064,A -85,B 0,C 180,E1 -20773.272,E2 -20773.272} C_VEL
LIN {X 0,Y 228.947,Z 359.826,A -85,B 0,C 180,E1 -20773.777,E2 -20773.777} C_VEL
LIN {X 0,Y 226.466,Z 427.253,A -85,B 0,C 180,E1 -20775.856,E2 -20775.856} C_VEL
LIN {X 0,Y 225.548,Z 440.445,A -85,B 0,C 180,E1 -20776.601,E2 -20776.601} C_VEL
LIN {X 0,Y 224.169,Z 453.189,A -85,B 0,C 180,E1 -20777.669,E2 -20777.669} C_VEL
LIN {X 0,Y 222.64,Z 465.266,A -85,B 0,C 180,E1 -20779.084,E2 -20779.084} C_VEL
LIN {X 0,Y 220.895,Z 476.758,A -85,B 0,C 180,E1 -20780.848,E2 -20780.848} C_VEL
LIN {X 0,Y 218.993,Z 487.15,A -85,B 0,C 180,E1 -20782.858,E2 -20782.858} C_VEL
LIN {X 0,Y 217.273,Z 495.653,A -85,B 0,C 180,E1 -20784.898,E2 -20784.898} C_VEL
LIN {X 0,Y 215.644,Z 503.486,A -85,B 0,C 180,E1 -20787.199,E2 -20787.199} C_VEL
LIN {X 0,Y 214.102,Z 511.128,A -85,B 0,C 180,E1 -20790.001,E2 -20790.001} C_VEL
LIN {X 0,Y 212.994,Z 517.268,A -85,B 0,C 180,E1 -20792.838,E2 -20792.838} C_VEL
LIN {X 0,Y 212.221,Z 522.142,A -85,B 0,C 180,E1 -20795.703,E2 -20795.703} C_VEL
LIN {X 0,Y 211.644,Z 525.901,A -85,B 0,C 180,E1 -20798.595,E2 -20798.595} C_VEL
LIN {X 0,Y 211.294,Z 528.629,A -85,B 0,C 180,E1 -20801.513,E2 -20801.513} C_VEL
LIN {X 0,Y 211.284,Z 529.915,A -85,B 0,C 180,E1 -20803.466,E2 -20803.466} C_VEL
LIN {X 0,Y 211.369,Z 530.774,A -85,B 0,C 180,E1 -20805.428,E2 -20805.428} C_VEL
LIN {X 0,Y 211.454,Z 531.198,A -85,B 0,C 180,E1 -20807.407,E2 -20807.407} C_VEL
LIN {X 0,Y 211.782,Z 531.22,A -85,B 0,C 180,E1 -20809.382,E2 -20809.382} C_VEL
LIN {X 0,Y 212.576,Z 530.499,A -85,B 0,C 180,E1 -20812.223,E2 -20812.223} C_VEL
LIN {X 0,Y 213.806,Z 528.713,A -85,B 0,C 180,E1 -20815.299,E2 -20815.299} C_VEL
LIN {X 0,Y 215.442,Z 525.92,A -85,B 0,C 180,E1 -20818.263,E2 -20818.263} C_VEL
LIN {X 0,Y 217.472,Z 522.087,A -85,B 0,C 180,E1 -20821.137,E2 -20821.137} C_VEL
LIN {X 0,Y 220.27,Z 516.505,A -85,B 0,C 180,E1 -20824.232,E2 -20824.232} C_VEL
LIN {X 0,Y 223.628,Z 509.238,A -85,B 0,C 180,E1 -20827.228,E2 -20827.228} C_VEL
LIN {X 0,Y 226.485,Z 502.461,A -85,B 0,C 180,E1 -20829.43,E2 -20829.43} C_VEL
LIN {X 0,Y 229.889,Z 493.777,A -85,B 0,C 180,E1 -20831.678,E2 -20831.678} C_VEL
LIN {X 0,Y 233.443,Z 483.66,A -85,B 0,C 180,E1 -20833.735,E2 -20833.735} C_VEL
LIN {X 0,Y 236.625,Z 472.755,A -85,B 0,C 180,E1 -20835.466,E2 -20835.466} C_VEL
LIN {X 0,Y 239.433,Z 461.133,A -85,B 0,C 180,E1 -20836.9,E2 -20836.9} C_VEL
LIN {X 0,Y 241.813,Z 448.623,A -85,B 0,C 180,E1 -20838.051,E2 -20838.051} C_VEL
LIN {X 0,Y 243.55,Z 435.372,A -85,B 0,C 180,E1 -20838.911,E2 -20838.911} C_VEL
LIN {X 0,Y 244.635,Z 422.058,A -85,B 0,C 180,E1 -20839.445,E2 -20839.445} C_VEL
LIN {X 0,Y 247.095,Z 378.152,A -85,B 0,C 180,E1 -20840.64,E2 -20840.64} C_VEL
LIN {X 0,Y 240.083,Z 363.575,A -85,B 0,C 180,E1 -20842.794,E2 -20842.794} C_VEL
LIN {X 0,Y 233.631,Z 352.27,A -85,B 0,C 180,E1 -20844.878,E2 -20844.878} C_VEL
LIN {X 0,Y 227.254,Z 342.738,A -85,B 0,C 180,E1 -20847.076,E2 -20847.076} C_VEL
LIN {X 0,Y 223.472,Z 337.656,A -85,B 0,C 180,E1 -20848.462,E2 -20848.462} C_VEL
LIN {X 0,Y 220.776,Z 333.884,A -85,B 0,C 180,E1 -20849.513,E2 -20849.513} C_VEL
LIN {X 0,Y 218.38,Z 330.925,A -85,B 0,C 180,E1 -20850.477,E2 -20850.477} C_VEL
LIN {X 0,Y 217.501,Z 329.22,A -85,B 0,C 180,E1 -20850.876,E2 -20850.876} C_VEL
LIN {X 0,Y 215.193,Z 327.255,A -85,B 0,C 180,E1 -20851.814,E2 -20851.814} C_VEL
LIN {X 0,Y 214.01,Z 324.821,A -85,B 0,C 180,E1 -20852.393,E2 -20852.393} C_VEL
LIN {X 0,Y 213.829,Z 323.842,A -85,B 0,C 180,E1 -20852.603,E2 -20852.603} C_VEL
LIN {X 0,Y 213.855,Z 323.834,A -85,B 0,C 180,E1 -20856.953,E2 -20856.953} C_VEL
LIN {X 0,Y 213.947,Z 323.831,A -85,B 0,C 180,E1 -20862.804,E2 -20862.804} C_VEL
LIN {X 0,Y 213.983,Z 323.819,A -85,B 0,C 180,E1 -20866.708,E2 -20866.708} C_VEL
LIN {X 0,Y 214.171,Z 323.789,A -85,B 0,C 180,E1 -20870.556,E2 -20870.556} C_VEL
LIN {X 0,Y 214.243,Z 323.794,A -85,B 0,C 180,E1 -20872.46,E2 -20872.46} C_VEL
LIN {X 0,Y 214.447,Z 323.772,A -85,B 0,C 180,E1 -20878.122,E2 -20878.122} C_VEL
LIN {X 0,Y 214.549,Z 323.743,A -85,B 0,C 180,E1 -20880,E2 -20880} C_VEL
LIN {X 0,Y 214.448,Z 323.755,A -85,B 0,C 180,E1 -20881.878,E2 -20881.878} C_VEL
LIN {X 0,Y 214.25,Z 323.784,A -85,B 0,C 180,E1 -20887.539,E2 -20887.539} C_VEL
LIN {X 0,Y 214.029,Z 323.804,A -85,B 0,C 180,E1 -20891.363,E2 -20891.363} C_VEL
LIN {X 0,Y 213.936,Z 323.823,A -85,B 0,C 180,E1 -20895.237,E2 -20895.237} C_VEL
LIN {X 0,Y 213.839,Z 323.847,A -85,B 0,C 180,E1 -20899.187,E2 -20899.187} C_VEL
LIN {X 0,Y 213.814,Z 323.852,A -85,B 0,C 180,E1 -20903.231,E2 -20903.231} C_VEL
LIN {X 0,Y 213.832,Z 323.846,A -85,B 0,C 180,E1 -20907.449,E2 -20907.449} C_VEL
LIN {X 0,Y 213.78,Z 323.854,A -85,B 0,C 180,E1 -20911.736,E2 -20911.736} C_VEL
LIN {X 0,Y 213.745,Z 323.854,A -85,B 0,C 180,E1 -20916.521,E2 -20916.521} C_VEL
LIN {X 0,Y 213.906,Z 324.491,A -85,B 0,C 180,E1 -20917.192,E2 -20917.192} C_VEL
LIN {X 0,Y 215.847,Z 330.477,A -85,B 0,C 180,E1 -20921.549,E2 -20921.549} C_VEL
LIN {X 0,Y 216.642,Z 332.375,A -85,B 0,C 180,E1 -20922.4,E2 -20922.4} C_VEL
LIN {X 0,Y 218.452,Z 336.463,A -85,B 0,C 180,E1 -20923.384,E2 -20923.384} C_VEL
LIN {X 0,Y 220.045,Z 341.328,A -85,B 0,C 180,E1 -20924.172,E2 -20924.172} C_VEL
LIN {X 0,Y 223.583,Z 353.705,A -85,B 0,C 180,E1 -20925.903,E2 -20925.903} C_VEL
LIN {X 0,Y 224.249,Z 355.323,A -85,B 0,C 180,E1 -20926.186,E2 -20926.186} C_VEL
LIN {X 0,Y 229.099,Z 363.996,A -85,B 0,C 180,E1 -20927.98,E2 -20927.98} C_VEL
LIN {X 0,Y 234.976,Z 375.914,A -85,B 0,C 180,E1 -20930.036,E2 -20930.036} C_VEL
LIN {X 0,Y 239.733,Z 387.04,A -85,B 0,C 180,E1 -20931.634,E2 -20931.634} C_VEL
LIN {X 0,Y 240.935,Z 396.709,A -85,B 0,C 180,E1 -20932.3,E2 -20932.3} C_VEL
LIN {X 0,Y 238.261,Z 442.632,A -85,B 0,C 180,E1 -20933.641,E2 -20933.641} C_VEL
LIN {X 0,Y 236.538,Z 456.279,A -85,B 0,C 180,E1 -20934.33,E2 -20934.33} C_VEL
LIN {X 0,Y 234.237,Z 468.523,A -85,B 0,C 180,E1 -20935.244,E2 -20935.244} C_VEL
LIN {X 0,Y 231.135,Z 481.089,A -85,B 0,C 180,E1 -20936.555,E2 -20936.555} C_VEL
LIN {X 0,Y 227.783,Z 492.297,A -85,B 0,C 180,E1 -20938.103,E2 -20938.103} C_VEL
LIN {X 0,Y 224.305,Z 502.426,A -85,B 0,C 180,E1 -20939.912,E2 -20939.912} C_VEL
LIN {X 0,Y 220.66,Z 511.567,A -85,B 0,C 180,E1 -20941.979,E2 -20941.979} C_VEL
LIN {X 0,Y 216.797,Z 520.487,A -85,B 0,C 180,E1 -20944.561,E2 -20944.561} C_VEL
LIN {X 0,Y 213.402,Z 528.095,A -85,B 0,C 180,E1 -20947.423,E2 -20947.423} C_VEL
LIN {X 0,Y 210.396,Z 534.307,A -85,B 0,C 180,E1 -20950.485,E2 -20950.485} C_VEL
LIN {X 0,Y 208.137,Z 538.714,A -85,B 0,C 180,E1 -20953.32,E2 -20953.32} C_VEL
LIN {X 0,Y 206.409,Z 542.073,A -85,B 0,C 180,E1 -20956.21,E2 -20956.21} C_VEL
LIN {X 0,Y 205.06,Z 545.06,A -85,B 0,C 180,E1 -20960.132,E2 -20960.132} C_VEL
LIN {X 0,Y 204.641,Z 545.969,A -85,B 0,C 180,E1 -20962.103,E2 -20962.103} C_VEL
LIN {X 0,Y 204.405,Z 546.552,A -85,B 0,C 180,E1 -20966.056,E2 -20966.056} C_VEL
LIN {X 0,Y 204.465,Z 546.266,A -85,B 0,C 180,E1 -20968.029,E2 -20968.029} C_VEL
LIN {X 0,Y 204.596,Z 545.592,A -85,B 0,C 180,E1 -20969.999,E2 -20969.999} C_VEL
LIN {X 0,Y 204.503,Z 544.477,A -85,B 0,C 180,E1 -20971.968,E2 -20971.968} C_VEL
LIN {X 0,Y 204.432,Z 542.444,A -85,B 0,C 180,E1 -20974.461,E2 -20974.461} C_VEL
LIN {X 0,Y 204.676,Z 538.497,A -85,B 0,C 180,E1 -20977.893,E2 -20977.893} C_VEL
LIN {X 0,Y 205.158,Z 533.859,A -85,B 0,C 180,E1 -20980.858,E2 -20980.858} C_VEL
LIN {X 0,Y 206.273,Z 526.816,A -85,B 0,C 180,E1 -20984.299,E2 -20984.299} C_VEL
LIN {X 0,Y 207.779,Z 519.18,A -85,B 0,C 180,E1 -20987.214,E2 -20987.214} C_VEL
LIN {X 0,Y 209.127,Z 513.025,A -85,B 0,C 180,E1 -20989.125,E2 -20989.125} C_VEL
LIN {X 0,Y 210.408,Z 506.216,A -85,B 0,C 180,E1 -20990.943,E2 -20990.943} C_VEL
LIN {X 0,Y 212.307,Z 496.136,A -85,B 0,C 180,E1 -20993.146,E2 -20993.146} C_VEL
LIN {X 0,Y 214.318,Z 485.556,A -85,B 0,C 180,E1 -20994.972,E2 -20994.972} C_VEL
LIN {X 0,Y 216.355,Z 473.882,A -85,B 0,C 180,E1 -20996.527,E2 -20996.527} C_VEL
LIN {X 0,Y 217.795,Z 462.998,A -85,B 0,C 180,E1 -20997.635,E2 -20997.635} C_VEL
LIN {X 0,Y 219.092,Z 450.261,A -85,B 0,C 180,E1 -20998.563,E2 -20998.563} C_VEL
LIN {X 0,Y 219.913,Z 436.953,A -85,B 0,C 180,E1 -20999.175,E2 -20999.175} C_VEL
LIN {X 0,Y 221.586,Z 389.135,A -85,B 0,C 180,E1 -21000.676,E2 -21000.676} C_VEL
LIN {X 0,Y 218.147,Z 357.929,A -85,B 0,C 180,E1 -21002.233,E2 -21002.233} C_VEL
LIN {X 0,Y 212.44,Z 342.787,A -85,B 0,C 180,E1 -21003.577,E2 -21003.577} C_VEL
LIN {X 0,Y 208.755,Z 333.63,A -85,B 0,C 180,E1 -21004.488,E2 -21004.488} C_VEL
LIN {X 0,Y 206.676,Z 324.738,A -85,B 0,C 180,E1 -21008.643,E2 -21008.643} C_VEL
LIN {X 0,Y 206.618,Z 324.746,A -85,B 0,C 180,E1 -21012.864,E2 -21012.864} C_VEL
LIN {X 0,Y 206.621,Z 324.747,A -85,B 0,C 180,E1 -21017.135,E2 -21017.135} C_VEL
LIN {X 0,Y 206.697,Z 324.735,A -85,B 0,C 180,E1 -21021.444,E2 -21021.444} C_VEL
LIN {X 0,Y 206.726,Z 324.732,A -85,B 0,C 180,E1 -21024.694,E2 -21024.694} C_VEL
LIN {X 0,Y 206.718,Z 324.734,A -85,B 0,C 180,E1 -21029.338,E2 -21029.338} C_VEL
LIN {X 0,Y 206.727,Z 324.732,A -85,B 0,C 180,E1 -21033.771,E2 -21033.771} C_VEL
LIN {X 0,Y 206.751,Z 324.73,A -85,B 0,C 180,E1 -21038.043,E2 -21038.043} C_VEL
LIN {X 0,Y 206.867,Z 324.697,A -85,B 0,C 180,E1 -21042.196,E2 -21042.196} C_VEL
LIN {X 0,Y 206.906,Z 324.707,A -85,B 0,C 180,E1 -21046.245,E2 -21046.245} C_VEL
LIN {X 0,Y 207.099,Z 324.682,A -85,B 0,C 180,E1 -21050.231,E2 -21050.231} C_VEL
LIN {X 0,Y 207.161,Z 324.664,A -85,B 0,C 180,E1 -21052.201,E2 -21052.201} C_VEL
LIN {X 0,Y 207.375,Z 324.651,A -85,B 0,C 180,E1 -21058.058,E2 -21058.058} C_VEL
LIN {X 0,Y 207.508,Z 324.635,A -85,B 0,C 180,E1 -21060,E2 -21060} C_VEL
LIN {X 0,Y 207.373,Z 324.647,A -85,B 0,C 180,E1 -21061.942,E2 -21061.942} C_VEL
LIN {X 0,Y 207.124,Z 324.664,A -85,B 0,C 180,E1 -21067.801,E2 -21067.801} C_VEL
LIN {X 0,Y 206.918,Z 324.709,A -85,B 0,C 180,E1 -21071.759,E2 -21071.759} C_VEL
LIN {X 0,Y 206.86,Z 324.711,A -85,B 0,C 180,E1 -21075.771,E2 -21075.771} C_VEL
LIN {X 0,Y 206.772,Z 324.729,A -85,B 0,C 180,E1 -21079.87,E2 -21079.87} C_VEL
LIN {X 0,Y 206.741,Z 324.731,A -85,B 0,C 180,E1 -21084.075,E2 -21084.075} C_VEL
LIN {X 0,Y 206.739,Z 324.726,A -85,B 0,C 180,E1 -21088.42,E2 -21088.42} C_VEL
LIN {X 0,Y 206.697,Z 324.73,A -85,B 0,C 180,E1 -21092.958,E2 -21092.958} C_VEL
LIN {X 0,Y 206.668,Z 324.737,A -85,B 0,C 180,E1 -21097.743,E2 -21097.743} C_VEL
LIN {X 0,Y 206.626,Z 324.744,A -85,B 0,C 180,E1 -21101.561,E2 -21101.561} C_VEL
LIN {X 0,Y 206.625,Z 324.745,A -85,B 0,C 180,E1 -21105.585,E2 -21105.585} C_VEL
LIN {X 0,Y 206.643,Z 324.743,A -85,B 0,C 180,E1 -21109.747,E2 -21109.747} C_VEL
LIN {X 0,Y 206.697,Z 324.737,A -85,B 0,C 180,E1 -21114.69,E2 -21114.69} C_VEL
LIN {X 0,Y 206.694,Z 324.738,A -85,B 0,C 180,E1 -21119.336,E2 -21119.336} C_VEL
LIN {X 0,Y 206.704,Z 324.737,A -85,B 0,C 180,E1 -21123.77,E2 -21123.77} C_VEL
LIN {X 0,Y 206.732,Z 324.728,A -85,B 0,C 180,E1 -21128.042,E2 -21128.042} C_VEL
LIN {X 0,Y 206.762,Z 324.784,A -85,B 0,C 180,E1 -21129.483,E2 -21129.483} C_VEL
LIN {X 0,Y 207.777,Z 327.549,A -85,B 0,C 180,E1 -21129.748,E2 -21129.748} C_VEL
LIN {X 0,Y 215.805,Z 343.242,A -85,B 0,C 180,E1 -21131.511,E2 -21131.511} C_VEL
LIN {X 0,Y 219.321,Z 352.097,A -85,B 0,C 180,E1 -21132.31,E2 -21132.31} C_VEL
LIN {X 0,Y 222.602,Z 361.848,A -85,B 0,C 180,E1 -21133.08,E2 -21133.08} C_VEL
LIN {X 0,Y 219.947,Z 427.575,A -85,B 0,C 180,E1 -21135.143,E2 -21135.143} C_VEL
LIN {X 0,Y 218.947,Z 441.361,A -85,B 0,C 180,E1 -21135.953,E2 -21135.953} C_VEL
LIN {X 0,Y 217.505,Z 453.943,A -85,B 0,C 180,E1 -21137.048,E2 -21137.048} C_VEL
LIN {X 0,Y 215.923,Z 465.876,A -85,B 0,C 180,E1 -21138.502,E2 -21138.502} C_VEL
LIN {X 0,Y 214.211,Z 476.807,A -85,B 0,C 180,E1 -21140.23,E2 -21140.23} C_VEL
LIN {X 0,Y 212.14,Z 487.651,A -85,B 0,C 180,E1 -21142.386,E2 -21142.386} C_VEL
LIN {X 0,Y 210.168,Z 496.941,A -85,B 0,C 180,E1 -21144.725,E2 -21144.725} C_VEL
LIN {X 0,Y 208.265,Z 505.948,A -85,B 0,C 180,E1 -21147.584,E2 -21147.584} C_VEL
LIN {X 0,Y 206.771,Z 513.204,A -85,B 0,C 180,E1 -21150.488,E2 -21150.488} C_VEL
LIN {X 0,Y 205.848,Z 518.095,A -85,B 0,C 180,E1 -21152.937,E2 -21152.937} C_VEL
LIN {X 0,Y 205.022,Z 523.315,A -85,B 0,C 180,E1 -21156.226,E2 -21156.226} C_VEL
LIN {X 0,Y 204.501,Z 526.502,A -85,B 0,C 180,E1 -21158.898,E2 -21158.898} C_VEL
LIN {X 0,Y 204.18,Z 529.127,A -85,B 0,C 180,E1 -21161.92,E2 -21161.92} C_VEL
LIN {X 0,Y 204.278,Z 531.016,A -85,B 0,C 180,E1 -21165.566,E2 -21165.566} C_VEL
LIN {X 0,Y 204.443,Z 531.496,A -85,B 0,C 180,E1 -21168.024,E2 -21168.024} C_VEL
LIN {X 0,Y 204.846,Z 531.467,A -85,B 0,C 180,E1 -21170.066,E2 -21170.066} C_VEL
LIN {X 0,Y 205.606,Z 530.787,A -85,B 0,C 180,E1 -21172.644,E2 -21172.644} C_VEL
LIN {X 0,Y 207.092,Z 528.756,A -85,B 0,C 180,E1 -21176.18,E2 -21176.18} C_VEL
LIN {X 0,Y 208.66,Z 526.25,A -85,B 0,C 180,E1 -21178.869,E2 -21178.869} C_VEL
LIN {X 0,Y 211.104,Z 521.907,A -85,B 0,C 180,E1 -21182.187,E2 -21182.187} C_VEL
LIN {X 0,Y 213.969,Z 516.523,A -85,B 0,C 180,E1 -21185.183,E2 -21185.183} C_VEL
LIN {X 0,Y 217.138,Z 510,A -85,B 0,C 180,E1 -21187.95,E2 -21187.95} C_VEL
LIN {X 0,Y 220.881,Z 501.588,A -85,B 0,C 180,E1 -21190.714,E2 -21190.714} C_VEL
LIN {X 0,Y 224.376,Z 492.911,A -85,B 0,C 180,E1 -21192.943,E2 -21192.943} C_VEL
LIN {X 0,Y 228.258,Z 482.079,A -85,B 0,C 180,E1 -21195.087,E2 -21195.087} C_VEL
LIN {X 0,Y 231.467,Z 471.218,A -85,B 0,C 180,E1 -21196.779,E2 -21196.779} C_VEL
LIN {X 0,Y 233.989,Z 461.016,A -85,B 0,C 180,E1 -21198.021,E2 -21198.021} C_VEL
LIN {X 0,Y 236.417,Z 448.711,A -85,B 0,C 180,E1 -21199.156,E2 -21199.156} C_VEL
LIN {X 0,Y 238.229,Z 435.362,A -85,B 0,C 180,E1 -21200.029,E2 -21200.029} C_VEL
LIN {X 0,Y 239.359,Z 421.82,A -85,B 0,C 180,E1 -21200.569,E2 -21200.569} C_VEL
LIN {X 0,Y 241.745,Z 380.515,A -85,B 0,C 180,E1 -21201.714,E2 -21201.714} C_VEL
LIN {X 0,Y 234.69,Z 365.909,A -85,B 0,C 180,E1 -21204.006,E2 -21204.006} C_VEL
LIN {X 0,Y 228.698,Z 355.456,A -85,B 0,C 180,E1 -21206.064,E2 -21206.064} C_VEL
LIN {X 0,Y 223.181,Z 347.479,A -85,B 0,C 180,E1 -21208.061,E2 -21208.061} C_VEL
LIN {X 0,Y 220.17,Z 343.232,A -85,B 0,C 180,E1 -21209.225,E2 -21209.225} C_VEL
LIN {X 0,Y 217.177,Z 339.133,A -85,B 0,C 180,E1 -21210.449,E2 -21210.449} C_VEL
LIN {X 0,Y 214.756,Z 335.695,A -85,B 0,C 180,E1 -21211.498,E2 -21211.498} C_VEL
LIN {X 0,Y 211.721,Z 332.277,A -85,B 0,C 180,E1 -21212.834,E2 -21212.834} C_VEL
LIN {X 0,Y 210.719,Z 330.247,A -85,B 0,C 180,E1 -21213.348,E2 -21213.348} C_VEL
LIN {X 0,Y 208.294,Z 328.34,A -85,B 0,C 180,E1 -21214.453,E2 -21214.453} C_VEL
LIN {X 0,Y 207.008,Z 325.876,A -85,B 0,C 180,E1 -21215.157,E2 -21215.157} C_VEL
LIN {X 0,Y 206.756,Z 324.729,A -85,B 0,C 180,E1 -21215.392,E2 -21215.392} C_VEL
LIN {X 0,Y 206.787,Z 324.716,A -85,B 0,C 180,E1 -21220.131,E2 -21220.131} C_VEL
LIN {X 0,Y 206.87,Z 324.708,A -85,B 0,C 180,E1 -21224.229,E2 -21224.229} C_VEL
LIN {X 0,Y 207.1,Z 324.672,A -85,B 0,C 180,E1 -21229.78,E2 -21229.78} C_VEL
LIN {X 0,Y 207.181,Z 324.67,A -85,B 0,C 180,E1 -21232.201,E2 -21232.201} C_VEL
LIN {X 0,Y 207.384,Z 324.651,A -85,B 0,C 180,E1 -21238.058,E2 -21238.058} C_VEL
LIN {X 0,Y 207.514,Z 324.619,A -85,B 0,C 180,E1 -21240,E2 -21240} C_VEL
LIN {X 0,Y 207.385,Z 324.635,A -85,B 0,C 180,E1 -21241.942,E2 -21241.942} C_VEL
LIN {X 0,Y 207.191,Z 324.666,A -85,B 0,C 180,E1 -21247.798,E2 -21247.798} C_VEL
LIN {X 0,Y 206.953,Z 324.686,A -85,B 0,C 180,E1 -21251.757,E2 -21251.757} C_VEL
LIN {X 0,Y 206.869,Z 324.7,A -85,B 0,C 180,E1 -21255.77,E2 -21255.77} C_VEL
LIN {X 0,Y 206.766,Z 324.72,A -85,B 0,C 180,E1 -21259.871,E2 -21259.871} C_VEL
LIN {X 0,Y 206.75,Z 324.727,A -85,B 0,C 180,E1 -21264.074,E2 -21264.074} C_VEL
LIN {X 0,Y 206.747,Z 324.728,A -85,B 0,C 180,E1 -21268.418,E2 -21268.418} C_VEL
LIN {X 0,Y 206.705,Z 324.728,A -85,B 0,C 180,E1 -21272.956,E2 -21272.956} C_VEL
LIN {X 0,Y 206.752,Z 324.878,A -85,B 0,C 180,E1 -21274.411,E2 -21274.411} C_VEL
LIN {X 0,Y 208.756,Z 331.095,A -85,B 0,C 180,E1 -21279.418,E2 -21279.418} C_VEL
LIN {X 0,Y 211.685,Z 335.756,A -85,B 0,C 180,E1 -21280.894,E2 -21280.894} C_VEL
LIN {X 0,Y 213.504,Z 338.19,A -85,B 0,C 180,E1 -21281.722,E2 -21281.722} C_VEL
LIN {X 0,Y 216.757,Z 342.946,A -85,B 0,C 180,E1 -21283.151,E2 -21283.151} C_VEL
LIN {X 0,Y 221.424,Z 350.613,A -85,B 0,C 180,E1 -21285.089,E2 -21285.089} C_VEL
LIN {X 0,Y 224.249,Z 355.323,A -85,B 0,C 180,E1 -21286.186,E2 -21286.186} C_VEL
LIN {X 0,Y 226.518,Z 361.846,A -85,B 0,C 180,E1 -21287.16,E2 -21287.16} C_VEL
LIN {X 0,Y 230.751,Z 379.619,A -85,B 0,C 180,E1 -21289.131,E2 -21289.131} C_VEL
LIN {X 0,Y 231.918,Z 382.961,A -85,B 0,C 180,E1 -21289.579,E2 -21289.579} C_VEL
LIN {X 0,Y 234.795,Z 389.941,A -85,B 0,C 180,E1 -21290.595,E2 -21290.595} C_VEL
LIN {X 0,Y 235.731,Z 397.551,A -85,B 0,C 180,E1 -21291.142,E2 -21291.142} C_VEL
LIN {X 0,Y 233.095,Z 441.69,A -85,B 0,C 180,E1 -21292.444,E2 -21292.444} C_VEL
LIN {X 0,Y 231.355,Z 455.375,A -85,B 0,C 180,E1 -21293.132,E2 -21293.132} C_VEL
LIN {X 0,Y 228.973,Z 467.804,A -85,B 0,C 180,E1 -21294.053,E2 -21294.053} C_VEL
LIN {X 0,Y 226.189,Z 478.921,A -85,B 0,C 180,E1 -21295.183,E2 -21295.183} C_VEL
LIN {X 0,Y 222.629,Z 490.476,A -85,B 0,C 180,E1 -21296.735,E2 -21296.735} C_VEL
LIN {X 0,Y 218.974,Z 500.884,A -85,B 0,C 180,E1 -21298.563,E2 -21298.563} C_VEL
LIN {X 0,Y 215.15,Z 510.297,A -85,B 0,C 180,E1 -21300.659,E2 -21300.659} C_VEL
LIN {X 0,Y 211.047,Z 519.387,A -85,B 0,C 180,E1 -21303.283,E2 -21303.283} C_VEL
LIN {X 0,Y 207.539,Z 526.735,A -85,B 0,C 180,E1 -21306.022,E2 -21306.022} C_VEL
LIN {X 0,Y 204.59,Z 532.661,A -85,B 0,C 180,E1 -21308.856,E2 -21308.856} C_VEL
LIN {X 0,Y 202.083,Z 537.369,A -85,B 0,C 180,E1 -21311.759,E2 -21311.759} C_VEL
LIN {X 0,Y 200.036,Z 540.992,A -85,B 0,C 180,E1 -21314.721,E2 -21314.721} C_VEL
LIN {X 0,Y 198.65,Z 543.634,A -85,B 0,C 180,E1 -21317.743,E2 -21317.743} C_VEL
LIN {X 0,Y 198.033,Z 544.9,A -85,B 0,C 180,E1 -21319.778,E2 -21319.778} C_VEL
LIN {X 0,Y 197.591,Z 545.761,A -85,B 0,C 180,E1 -21321.819,E2 -21321.819} C_VEL
LIN {X 0,Y 197.326,Z 546.272,A -85,B 0,C 180,E1 -21325.914,E2 -21325.914} C_VEL
LIN {X 0,Y 197.365,Z 545.954,A -85,B 0,C 180,E1 -21327.958,E2 -21327.958} C_VEL
LIN {X 0,Y 197.51,Z 545.246,A -85,B 0,C 180,E1 -21329.999,E2 -21329.999} C_VEL
LIN {X 0,Y 197.401,Z 544.074,A -85,B 0,C 180,E1 -21332.039,E2 -21332.039} C_VEL
LIN {X 0,Y 197.343,Z 542.28,A -85,B 0,C 180,E1 -21334.313,E2 -21334.313} C_VEL
LIN {X 0,Y 197.499,Z 539.26,A -85,B 0,C 180,E1 -21337.153,E2 -21337.153} C_VEL
LIN {X 0,Y 197.933,Z 534.94,A -85,B 0,C 180,E1 -21340.225,E2 -21340.225} C_VEL
LIN {X 0,Y 198.737,Z 529.398,A -85,B 0,C 180,E1 -21343.287,E2 -21343.287} C_VEL
LIN {X 0,Y 200.167,Z 522.472,A -85,B 0,C 180,E1 -21346.311,E2 -21346.311} C_VEL
LIN {X 0,Y 201.705,Z 515.382,A -85,B 0,C 180,E1 -21348.8,E2 -21348.8} C_VEL
LIN {X 0,Y 202.999,Z 508.52,A -85,B 0,C 180,E1 -21350.809,E2 -21350.809} C_VEL
LIN {X 0,Y 204.899,Z 499.607,A -85,B 0,C 180,E1 -21352.963,E2 -21352.963} C_VEL
LIN {X 0,Y 206.863,Z 489.886,A -85,B 0,C 180,E1 -21354.86,E2 -21354.86} C_VEL
LIN {X 0,Y 208.713,Z 479.398,A -85,B 0,C 180,E1 -21356.496,E2 -21356.496} C_VEL
LIN {X 0,Y 210.48,Z 467.925,A -85,B 0,C 180,E1 -21357.868,E2 -21357.868} C_VEL
LIN {X 0,Y 212.082,Z 455.009,A -85,B 0,C 180,E1 -21358.987,E2 -21358.987} C_VEL
LIN {X 0,Y 213.186,Z 442.305,A -85,B 0,C 180,E1 -21359.72,E2 -21359.72} C_VEL
LIN {X 0,Y 215.128,Z 389.276,A -85,B 0,C 180,E1 -21361.475,E2 -21361.475} C_VEL
LIN {X 0,Y 211.873,Z 359.786,A -85,B 0,C 180,E1 -21363.014,E2 -21363.014} C_VEL
LIN {X 0,Y 205.974,Z 344.184,A -85,B 0,C 180,E1 -21364.475,E2 -21364.475} C_VEL
LIN {X 0,Y 201.422,Z 333.26,A -85,B 0,C 180,E1 -21365.678,E2 -21365.678} C_VEL
LIN {X 0,Y 199.621,Z 325.615,A -85,B 0,C 180,E1 -21369.486,E2 -21369.486} C_VEL
LIN {X 0,Y 199.574,Z 325.626,A -85,B 0,C 180,E1 -21374.77,E2 -21374.77} C_VEL
LIN {X 0,Y 199.578,Z 325.625,A -85,B 0,C 180,E1 -21378.005,E2 -21378.005} C_VEL
LIN {X 0,Y 199.636,Z 325.61,A -85,B 0,C 180,E1 -21380.755,E2 -21380.755} C_VEL
LIN {X 0,Y 199.63,Z 325.616,A -85,B 0,C 180,E1 -21385.717,E2 -21385.717} C_VEL
LIN {X 0,Y 199.699,Z 325.605,A -85,B 0,C 180,E1 -21388.137,E2 -21388.137} C_VEL
LIN {X 0,Y 199.681,Z 325.611,A -85,B 0,C 180,E1 -21392.771,E2 -21392.771} C_VEL
LIN {X 0,Y 199.732,Z 325.607,A -85,B 0,C 180,E1 -21397.228,E2 -21397.228} C_VEL
LIN {X 0,Y 199.79,Z 325.58,A -85,B 0,C 180,E1 -21401.757,E2 -21401.757} C_VEL
LIN {X 0,Y 199.84,Z 325.586,A -85,B 0,C 180,E1 -21405.749,E2 -21405.749} C_VEL
LIN {X 0,Y 200.064,Z 325.559,A -85,B 0,C 180,E1 -21409.884,E2 -21409.884} C_VEL
LIN {X 0,Y 200.027,Z 325.541,A -85,B 0,C 180,E1 -21413.95,E2 -21413.95} C_VEL
LIN {X 0,Y 200.315,Z 325.529,A -85,B 0,C 180,E1 -21417.989,E2 -21417.989} C_VEL
LIN {X 0,Y 200.472,Z 325.512,A -85,B 0,C 180,E1 -21420,E2 -21420} C_VEL
LIN {X 0,Y 200.013,Z 325.551,A -85,B 0,C 180,E1 -21424.03,E2 -21424.03} C_VEL
LIN {X 0,Y 200.072,Z 325.543,A -85,B 0,C 180,E1 -21428.077,E2 -21428.077} C_VEL
LIN {X 0,Y 199.868,Z 325.589,A -85,B 0,C 180,E1 -21432.18,E2 -21432.18} C_VEL
LIN {X 0,Y 199.798,Z 325.593,A -85,B 0,C 180,E1 -21436.344,E2 -21436.344} C_VEL
LIN {X 0,Y 199.684,Z 325.606,A -85,B 0,C 180,E1 -21440.607,E2 -21440.607} C_VEL
LIN {X 0,Y 199.659,Z 325.613,A -85,B 0,C 180,E1 -21444.986,E2 -21444.986} C_VEL
LIN {X 0,Y 199.669,Z 325.609,A -85,B 0,C 180,E1 -21449.523,E2 -21449.523} C_VEL
LIN {X 0,Y 199.672,Z 325.609,A -85,B 0,C 180,E1 -21452.359,E2 -21452.359} C_VEL
LIN {X 0,Y 199.615,Z 325.619,A -85,B 0,C 180,E1 -21456.765,E2 -21456.765} C_VEL
LIN {X 0,Y 199.59,Z 325.616,A -85,B 0,C 180,E1 -21459.333,E2 -21459.333} C_VEL
LIN {X 0,Y 199.561,Z 325.625,A -85,B 0,C 180,E1 -21462.309,E2 -21462.309} C_VEL
LIN {X 0,Y 199.571,Z 325.623,A -85,B 0,C 180,E1 -21465.229,E2 -21465.229} C_VEL
LIN {X 0,Y 199.566,Z 325.622,A -85,B 0,C 180,E1 -21468.004,E2 -21468.004} C_VEL
LIN {X 0,Y 199.593,Z 325.623,A -85,B 0,C 180,E1 -21470.774,E2 -21470.774} C_VEL
LIN {X 0,Y 199.608,Z 325.62,A -85,B 0,C 180,E1 -21475.715,E2 -21475.715} C_VEL
LIN {X 0,Y 199.683,Z 325.611,A -85,B 0,C 180,E1 -21478.136,E2 -21478.136} C_VEL
LIN {X 0,Y 199.642,Z 325.617,A -85,B 0,C 180,E1 -21482.767,E2 -21482.767} C_VEL
LIN {X 0,Y 199.706,Z 325.609,A -85,B 0,C 180,E1 -21487.227,E2 -21487.227} C_VEL
LIN {X 0,Y 199.711,Z 325.601,A -85,B 0,C 180,E1 -21488.369,E2 -21488.369} C_VEL
LIN {X 0,Y 200.722,Z 328.46,A -85,B 0,C 180,E1 -21488.663,E2 -21488.663} C_VEL
LIN {X 0,Y 208.058,Z 342.394,A -85,B 0,C 180,E1 -21490.369,E2 -21490.369} C_VEL
LIN {X 0,Y 212.106,Z 351.497,A -85,B 0,C 180,E1 -21491.306,E2 -21491.306} C_VEL
LIN {X 0,Y 216.078,Z 362.757,A -85,B 0,C 180,E1 -21492.272,E2 -21492.272} C_VEL
LIN {X 0,Y 213.43,Z 428.199,A -85,B 0,C 180,E1 -21494.4,E2 -21494.4} C_VEL
LIN {X 0,Y 212.439,Z 441.514,A -85,B 0,C 180,E1 -21495.207,E2 -21495.207} C_VEL
LIN {X 0,Y 210.868,Z 454.662,A -85,B 0,C 180,E1 -21496.387,E2 -21496.387} C_VEL
LIN {X 0,Y 209.229,Z 466.477,A -85,B 0,C 180,E1 -21497.883,E2 -21497.883} C_VEL
LIN {X 0,Y 207.416,Z 477.577,A -85,B 0,C 180,E1 -21499.704,E2 -21499.704} C_VEL
LIN {X 0,Y 205.307,Z 488.133,A -85,B 0,C 180,E1 -21501.884,E2 -21501.884} C_VEL
LIN {X 0,Y 203.056,Z 498.2,A -85,B 0,C 180,E1 -21504.54,E2 -21504.54} C_VEL
LIN {X 0,Y 201.13,Z 507.04,A -85,B 0,C 180,E1 -21507.498,E2 -21507.498} C_VEL
LIN {X 0,Y 199.634,Z 514.102,A -85,B 0,C 180,E1 -21510.506,E2 -21510.506} C_VEL
LIN {X 0,Y 198.419,Z 520.562,A -85,B 0,C 180,E1 -21514.064,E2 -21514.064} C_VEL
LIN {X 0,Y 197.707,Z 524.825,A -85,B 0,C 180,E1 -21517.147,E2 -21517.147} C_VEL
LIN {X 0,Y 197.205,Z 528.026,A -85,B 0,C 180,E1 -21520.266,E2 -21520.266} C_VEL
LIN {X 0,Y 197.082,Z 529.62,A -85,B 0,C 180,E1 -21522.356,E2 -21522.356} C_VEL
LIN {X 0,Y 197.18,Z 531.27,A -85,B 0,C 180,E1 -21525.771,E2 -21525.771} C_VEL
LIN {X 0,Y 197.444,Z 531.794,A -85,B 0,C 180,E1 -21528.686,E2 -21528.686} C_VEL
LIN {X 0,Y 197.923,Z 531.697,A -85,B 0,C 180,E1 -21530.8,E2 -21530.8} C_VEL
LIN {X 0,Y 198.658,Z 531.071,A -85,B 0,C 180,E1 -21533.101,E2 -21533.101} C_VEL
LIN {X 0,Y 200.429,Z 528.798,A -85,B 0,C 180,E1 -21537.12,E2 -21537.12} C_VEL
LIN {X 0,Y 202.423,Z 525.779,A -85,B 0,C 180,E1 -21540.27,E2 -21540.27} C_VEL
LIN {X 0,Y 204.836,Z 521.713,A -85,B 0,C 180,E1 -21543.297,E2 -21543.297} C_VEL
LIN {X 0,Y 208.326,Z 515.394,A -85,B 0,C 180,E1 -21546.725,E2 -21546.725} C_VEL
LIN {X 0,Y 211.836,Z 508.393,A -85,B 0,C 180,E1 -21549.608,E2 -21549.608} C_VEL
LIN {X 0,Y 215.306,Z 500.925,A -85,B 0,C 180,E1 -21552.003,E2 -21552.003} C_VEL
LIN {X 0,Y 219.038,Z 491.996,A -85,B 0,C 180,E1 -21554.257,E2 -21554.257} C_VEL
LIN {X 0,Y 222.514,Z 482.579,A -85,B 0,C 180,E1 -21556.137,E2 -21556.137} C_VEL
LIN {X 0,Y 226.008,Z 471.201,A -85,B 0,C 180,E1 -21557.939,E2 -21557.939} C_VEL
LIN {X 0,Y 229.075,Z 458.924,A -85,B 0,C 180,E1 -21559.406,E2 -21559.406} C_VEL
LIN {X 0,Y 231.462,Z 446.682,A -85,B 0,C 180,E1 -21560.478,E2 -21560.478} C_VEL
LIN {X 0,Y 233.163,Z 433.641,A -85,B 0,C 180,E1 -21561.301,E2 -21561.301} C_VEL
LIN {X 0,Y 234.318,Z 419.162,A -85,B 0,C 180,E1 -21561.815,E2 -21561.815} C_VEL
LIN {X 0,Y 236.476,Z 382.86,A -85,B 0,C 180,E1 -21562.839,E2 -21562.839} C_VEL
LIN {X 0,Y 230.03,Z 369.574,A -85,B 0,C 180,E1 -21565.05,E2 -21565.05} C_VEL
LIN {X 0,Y 225.015,Z 360.677,A -85,B 0,C 180,E1 -21566.867,E2 -21566.867} C_VEL
LIN {X 0,Y 219.103,Z 351.937,A -85,B 0,C 180,E1 -21569.121,E2 -21569.121} C_VEL
LIN {X 0,Y 214.296,Z 345.124,A -85,B 0,C 180,E1 -21571.137,E2 -21571.137} C_VEL
LIN {X 0,Y 211.056,Z 340.8,A -85,B 0,C 180,E1 -21572.591,E2 -21572.591} C_VEL
LIN {X 0,Y 208.476,Z 337.473,A -85,B 0,C 180,E1 -21573.814,E2 -21573.814} C_VEL
LIN {X 0,Y 207.534,Z 336.156,A -85,B 0,C 180,E1 -21574.285,E2 -21574.285} C_VEL
LIN {X 0,Y 205.071,Z 333.518,A -85,B 0,C 180,E1 -21575.514,E2 -21575.514} C_VEL
LIN {X 0,Y 203.819,Z 331.174,A -85,B 0,C 180,E1 -21576.234,E2 -21576.234} C_VEL
LIN {X 0,Y 201.314,Z 329.257,A -85,B 0,C 180,E1 -21577.552,E2 -21577.552} C_VEL
LIN {X 0,Y 200.043,Z 327.038,A -85,B 0,C 180,E1 -21578.353,E2 -21578.353} C_VEL
LIN {X 0,Y 199.698,Z 325.608,A -85,B 0,C 180,E1 -21578.72,E2 -21578.72} C_VEL
LIN {X 0,Y 199.8,Z 325.583,A -85,B 0,C 180,E1 -21581.758,E2 -21581.758} C_VEL
LIN {X 0,Y 199.851,Z 325.574,A -85,B 0,C 180,E1 -21585.749,E2 -21585.749} C_VEL
LIN {X 0,Y 200.074,Z 325.547,A -85,B 0,C 180,E1 -21589.884,E2 -21589.884} C_VEL
LIN {X 0,Y 200.039,Z 325.561,A -85,B 0,C 180,E1 -21593.95,E2 -21593.95} C_VEL
LIN {X 0,Y 200.323,Z 325.53,A -85,B 0,C 180,E1 -21597.989,E2 -21597.989} C_VEL
LIN {X 0,Y 200.479,Z 325.494,A -85,B 0,C 180,E1 -21600,E2 -21600} C_VEL
LIN {X 0,Y 200.034,Z 325.562,A -85,B 0,C 180,E1 -21604.029,E2 -21604.029} C_VEL
LIN {X 0,Y 200.135,Z 325.548,A -85,B 0,C 180,E1 -21608.075,E2 -21608.075} C_VEL
LIN {X 0,Y 199.896,Z 325.567,A -85,B 0,C 180,E1 -21612.178,E2 -21612.178} C_VEL
LIN {X 0,Y 199.807,Z 325.578,A -85,B 0,C 180,E1 -21616.343,E2 -21616.343} C_VEL
LIN {X 0,Y 199.685,Z 325.596,A -85,B 0,C 180,E1 -21620.607,E2 -21620.607} C_VEL
LIN {X 0,Y 199.667,Z 325.601,A -85,B 0,C 180,E1 -21624.985,E2 -21624.985} C_VEL
LIN {X 0,Y 199.678,Z 325.599,A -85,B 0,C 180,E1 -21629.522,E2 -21629.522} C_VEL
LIN {X 0,Y 199.711,Z 325.705,A -85,B 0,C 180,E1 -21631.565,E2 -21631.565} C_VEL
LIN {X 0,Y 200.615,Z 328.329,A -85,B 0,C 180,E1 -21634.091,E2 -21634.091} C_VEL
LIN {X 0,Y 201.415,Z 330.788,A -85,B 0,C 180,E1 -21636.143,E2 -21636.143} C_VEL
LIN {X 0,Y 204.509,Z 335.43,A -85,B 0,C 180,E1 -21637.9,E2 -21637.9} C_VEL
LIN {X 0,Y 206.242,Z 337.659,A -85,B 0,C 180,E1 -21638.802,E2 -21638.802} C_VEL
LIN {X 0,Y 209.804,Z 342.781,A -85,B 0,C 180,E1 -21640.577,E2 -21640.577} C_VEL
LIN {X 0,Y 213.603,Z 348.583,A -85,B 0,C 180,E1 -21642.345,E2 -21642.345} C_VEL
LIN {X 0,Y 218.279,Z 356.446,A -85,B 0,C 180,E1 -21644.383,E2 -21644.383} C_VEL
LIN {X 0,Y 223.412,Z 365.496,A -85,B 0,C 180,E1 -21646.433,E2 -21646.433} C_VEL
LIN {X 0,Y 228.707,Z 375.933,A -85,B 0,C 180,E1 -21648.423,E2 -21648.423} C_VEL
LIN {X 0,Y 231.918,Z 382.961,A -85,B 0,C 180,E1 -21649.579,E2 -21649.579} C_VEL
LIN {X 0,Y 232.818,Z 386.416,A -85,B 0,C 180,E1 -21649.957,E2 -21649.957} C_VEL
LIN {X 0,Y 233.098,Z 390.198,A -85,B 0,C 180,E1 -21650.191,E2 -21650.191} C_VEL
LIN {X 0,Y 232.909,Z 394.146,A -85,B 0,C 180,E1 -21650.316,E2 -21650.316} C_VEL
LIN {X 0,Y 232.392,Z 398.1,A -85,B 0,C 180,E1 -21650.36,E2 -21650.36} C_VEL
LIN {X 0,Y 230.176,Z 410.5,A -85,B 0,C 180,E1 -21650.353,E2 -21650.353} C_VEL
LIN {X 0,Y 229.742,Z 414.651,A -85,B 0,C 180,E1 -21650.427,E2 -21650.427} C_VEL
LIN {X 0,Y 227.843,Z 442.674,A -85,B 0,C 180,E1 -21651.278,E2 -21651.278} C_VEL
LIN {X 0,Y 226.021,Z 455.979,A -85,B 0,C 180,E1 -21651.97,E2 -21651.97} C_VEL
LIN {X 0,Y 223.558,Z 468.148,A -85,B 0,C 180,E1 -21652.9,E2 -21652.9} C_VEL
LIN {X 0,Y 220.45,Z 479.893,A -85,B 0,C 180,E1 -21654.139,E2 -21654.139} C_VEL
LIN {X 0,Y 216.765,Z 491.224,A -85,B 0,C 180,E1 -21655.712,E2 -21655.712} C_VEL
LIN {X 0,Y 212.979,Z 501.456,A -85,B 0,C 180,E1 -21657.572,E2 -21657.572} C_VEL
LIN {X 0,Y 209.022,Z 510.68,A -85,B 0,C 180,E1 -21659.711,E2 -21659.711} C_VEL
LIN {X 0,Y 204.742,Z 519.654,A -85,B 0,C 180,E1 -21662.392,E2 -21662.392} C_VEL
LIN {X 0,Y 201.06,Z 526.908,A -85,B 0,C 180,E1 -21665.199,E2 -21665.199} C_VEL
LIN {X 0,Y 197.978,Z 532.747,A -85,B 0,C 180,E1 -21668.114,E2 -21668.114} C_VEL
LIN {X 0,Y 195.353,Z 537.377,A -85,B 0,C 180,E1 -21671.107,E2 -21671.107} C_VEL
LIN {X 0,Y 193.16,Z 540.929,A -85,B 0,C 180,E1 -21674.163,E2 -21674.163} C_VEL
LIN {X 0,Y 191.69,Z 543.506,A -85,B 0,C 180,E1 -21677.291,E2 -21677.291} C_VEL
LIN {X 0,Y 191.026,Z 544.738,A -85,B 0,C 180,E1 -21679.398,E2 -21679.398} C_VEL
LIN {X 0,Y 190.293,Z 545.955,A -85,B 0,C 180,E1 -21683.637,E2 -21683.637} C_VEL
LIN {X 0,Y 190.236,Z 545.981,A -85,B 0,C 180,E1 -21685.932,E2 -21685.932} C_VEL
LIN {X 0,Y 190.425,Z 544.882,A -85,B 0,C 180,E1 -21689.998,E2 -21689.998} C_VEL
LIN {X 0,Y 190.301,Z 543.67,A -85,B 0,C 180,E1 -21692.115,E2 -21692.115} C_VEL
LIN {X 0,Y 190.266,Z 541.068,A -85,B 0,C 180,E1 -21695.297,E2 -21695.297} C_VEL
LIN {X 0,Y 190.564,Z 537.427,A -85,B 0,C 180,E1 -21698.482,E2 -21698.482} C_VEL
LIN {X 0,Y 191.163,Z 532.636,A -85,B 0,C 180,E1 -21701.664,E2 -21701.664} C_VEL
LIN {X 0,Y 192.208,Z 526.557,A -85,B 0,C 180,E1 -21704.828,E2 -21704.828} C_VEL
LIN {X 0,Y 193.839,Z 518.979,A -85,B 0,C 180,E1 -21707.948,E2 -21707.948} C_VEL
LIN {X 0,Y 195.407,Z 511.827,A -85,B 0,C 180,E1 -21710.325,E2 -21710.325} C_VEL
LIN {X 0,Y 197.695,Z 501.779,A -85,B 0,C 180,E1 -21713.018,E2 -21713.018} C_VEL
LIN {X 0,Y 199.594,Z 492.545,A -85,B 0,C 180,E1 -21714.993,E2 -21714.993} C_VEL
LIN {X 0,Y 201.719,Z 481.111,A -85,B 0,C 180,E1 -21716.93,E2 -21716.93} C_VEL
LIN {X 0,Y 203.578,Z 470.27,A -85,B 0,C 180,E1 -21718.337,E2 -21718.337} C_VEL
LIN {X 0,Y 205.178,Z 458.453,A -85,B 0,C 180,E1 -21719.496,E2 -21719.496} C_VEL
LIN {X 0,Y 206.52,Z 445.733,A -85,B 0,C 180,E1 -21720.339,E2 -21720.339} C_VEL
LIN {X 0,Y 207.369,Z 429.049,A -85,B 0,C 180,E1 -21720.992,E2 -21720.992} C_VEL
LIN {X 0,Y 208.721,Z 389.589,A -85,B 0,C 180,E1 -21722.316,E2 -21722.316} C_VEL
LIN {X 0,Y 205.767,Z 362.034,A -85,B 0,C 180,E1 -21723.806,E2 -21723.806} C_VEL
LIN {X 0,Y 199.382,Z 345.283,A -85,B 0,C 180,E1 -21725.47,E2 -21725.47} C_VEL
LIN {X 0,Y 194.143,Z 333.078,A -85,B 0,C 180,E1 -21726.874,E2 -21726.874} C_VEL
LIN {X 0,Y 192.579,Z 326.495,A -85,B 0,C 180,E1 -21730.267,E2 -21730.267} C_VEL
LIN {X 0,Y 192.487,Z 326.509,A -85,B 0,C 180,E1 -21736.075,E2 -21736.075} C_VEL
LIN {X 0,Y 192.536,Z 326.493,A -85,B 0,C 180,E1 -21740.042,E2 -21740.042} C_VEL
LIN {X 0,Y 192.593,Z 326.492,A -85,B 0,C 180,E1 -21744.277,E2 -21744.277} C_VEL
LIN {X 0,Y 192.602,Z 326.493,A -85,B 0,C 180,E1 -21749.279,E2 -21749.279} C_VEL
LIN {X 0,Y 192.659,Z 326.483,A -85,B 0,C 180,E1 -21751.691,E2 -21751.691} C_VEL
LIN {X 0,Y 192.7,Z 326.478,A -85,B 0,C 180,E1 -21756.348,E2 -21756.348} C_VEL
LIN {X 0,Y 192.726,Z 326.46,A -85,B 0,C 180,E1 -21761.457,E2 -21761.457} C_VEL
LIN {X 0,Y 192.764,Z 326.462,A -85,B 0,C 180,E1 -21765.214,E2 -21765.214} C_VEL
LIN {X 0,Y 192.975,Z 326.444,A -85,B 0,C 180,E1 -21769.508,E2 -21769.508} C_VEL
LIN {X 0,Y 193.055,Z 326.422,A -85,B 0,C 180,E1 -21771.627,E2 -21771.627} C_VEL
LIN {X 0,Y 193.257,Z 326.407,A -85,B 0,C 180,E1 -21777.916,E2 -21777.916} C_VEL
LIN {X 0,Y 193.436,Z 326.388,A -85,B 0,C 180,E1 -21780,E2 -21780} C_VEL
LIN {X 0,Y 192.959,Z 326.428,A -85,B 0,C 180,E1 -21784.178,E2 -21784.178} C_VEL
LIN {X 0,Y 193.021,Z 326.423,A -85,B 0,C 180,E1 -21788.375,E2 -21788.375} C_VEL
LIN {X 0,Y 192.796,Z 326.468,A -85,B 0,C 180,E1 -21792.634,E2 -21792.634} C_VEL
LIN {X 0,Y 192.751,Z 326.472,A -85,B 0,C 180,E1 -21796.959,E2 -21796.959} C_VEL
LIN {X 0,Y 192.615,Z 326.485,A -85,B 0,C 180,E1 -21801.4,E2 -21801.4} C_VEL
LIN {X 0,Y 192.641,Z 326.488,A -85,B 0,C 180,E1 -21804.214,E2 -21804.214} C_VEL
LIN {X 0,Y 192.645,Z 326.483,A -85,B 0,C 180,E1 -21808.893,E2 -21808.893} C_VEL
LIN {X 0,Y 192.594,Z 326.486,A -85,B 0,C 180,E1 -21813.187,E2 -21813.187} C_VEL
LIN {X 0,Y 192.538,Z 326.496,A -85,B 0,C 180,E1 -21818.355,E2 -21818.355} C_VEL
LIN {X 0,Y 192.48,Z 326.504,A -85,B 0,C 180,E1 -21823.095,E2 -21823.095} C_VEL
LIN {X 0,Y 192.481,Z 326.509,A -85,B 0,C 180,E1 -21826.908,E2 -21826.908} C_VEL
LIN {X 0,Y 192.538,Z 326.5,A -85,B 0,C 180,E1 -21831.648,E2 -21831.648} C_VEL
LIN {X 0,Y 192.592,Z 326.492,A -85,B 0,C 180,E1 -21836.815,E2 -21836.815} C_VEL
LIN {X 0,Y 192.619,Z 326.493,A -85,B 0,C 180,E1 -21841.687,E2 -21841.687} C_VEL
LIN {X 0,Y 192.679,Z 326.543,A -85,B 0,C 180,E1 -21847.186,E2 -21847.186} C_VEL
LIN {X 0,Y 193.664,Z 329.327,A -85,B 0,C 180,E1 -21847.484,E2 -21847.484} C_VEL
LIN {X 0,Y 197.863,Z 336.898,A -85,B 0,C 180,E1 -21848.535,E2 -21848.535} C_VEL
LIN {X 0,Y 205.292,Z 351.963,A -85,B 0,C 180,E1 -21850.33,E2 -21850.33} C_VEL
LIN {X 0,Y 209.683,Z 364.268,A -85,B 0,C 180,E1 -21851.45,E2 -21851.45} C_VEL
LIN {X 0,Y 207.815,Z 411.573,A -85,B 0,C 180,E1 -21853.002,E2 -21853.002} C_VEL
LIN {X 0,Y 206.841,Z 430.961,A -85,B 0,C 180,E1 -21853.723,E2 -21853.723} C_VEL
LIN {X 0,Y 205.839,Z 443.173,A -85,B 0,C 180,E1 -21854.531,E2 -21854.531} C_VEL
LIN {X 0,Y 204.261,Z 455.358,A -85,B 0,C 180,E1 -21855.684,E2 -21855.684} C_VEL
LIN {X 0,Y 202.561,Z 467.078,A -85,B 0,C 180,E1 -21857.223,E2 -21857.223} C_VEL
LIN {X 0,Y 200.64,Z 478.34,A -85,B 0,C 180,E1 -21859.142,E2 -21859.142} C_VEL
LIN {X 0,Y 198.487,Z 488.612,A -85,B 0,C 180,E1 -21861.347,E2 -21861.347} C_VEL
LIN {X 0,Y 196.361,Z 497.816,A -85,B 0,C 180,E1 -21863.838,E2 -21863.838} C_VEL
LIN {X 0,Y 194.316,Z 506.765,A -85,B 0,C 180,E1 -21866.892,E2 -21866.892} C_VEL
LIN {X 0,Y 192.701,Z 513.963,A -85,B 0,C 180,E1 -21870.002,E2 -21870.002} C_VEL
LIN {X 0,Y 191.539,Z 519.692,A -85,B 0,C 180,E1 -21873.157,E2 -21873.157} C_VEL
LIN {X 0,Y 190.776,Z 524.207,A -85,B 0,C 180,E1 -21876.347,E2 -21876.347} C_VEL
LIN {X 0,Y 190.354,Z 526.605,A -85,B 0,C 180,E1 -21878.494,E2 -21878.494} C_VEL
LIN {X 0,Y 190.088,Z 528.57,A -85,B 0,C 180,E1 -21880.654,E2 -21880.654} C_VEL
LIN {X 0,Y 189.973,Z 530.082,A -85,B 0,C 180,E1 -21882.826,E2 -21882.826} C_VEL
LIN {X 0,Y 190.104,Z 531.53,A -85,B 0,C 180,E1 -21886.012,E2 -21886.012} C_VEL
LIN {X 0,Y 190.495,Z 532.087,A -85,B 0,C 180,E1 -21889.394,E2 -21889.394} C_VEL
LIN {X 0,Y 191.693,Z 531.365,A -85,B 0,C 180,E1 -21893.57,E2 -21893.57} C_VEL
LIN {X 0,Y 192.68,Z 530.277,A -85,B 0,C 180,E1 -21895.958,E2 -21895.958} C_VEL
LIN {X 0,Y 193.844,Z 528.802,A -85,B 0,C 180,E1 -21898.122,E2 -21898.122} C_VEL
LIN {X 0,Y 195.986,Z 525.716,A -85,B 0,C 180,E1 -21901.331,E2 -21901.331} C_VEL
LIN {X 0,Y 198.653,Z 521.485,A -85,B 0,C 180,E1 -21904.477,E2 -21904.477} C_VEL
LIN {X 0,Y 202.471,Z 514.937,A -85,B 0,C 180,E1 -21908.035,E2 -21908.035} C_VEL
LIN {X 0,Y 205.571,Z 509,A -85,B 0,C 180,E1 -21910.51,E2 -21910.51} C_VEL
LIN {X 0,Y 209.095,Z 501.818,A -85,B 0,C 180,E1 -21912.894,E2 -21912.894} C_VEL
LIN {X 0,Y 212.966,Z 493.076,A -85,B 0,C 180,E1 -21915.196,E2 -21915.196} C_VEL
LIN {X 0,Y 216.821,Z 483.165,A -85,B 0,C 180,E1 -21917.227,E2 -21917.227} C_VEL
LIN {X 0,Y 220.211,Z 472.671,A -85,B 0,C 180,E1 -21918.938,E2 -21918.938} C_VEL
LIN {X 0,Y 223.398,Z 460.846,A -85,B 0,C 180,E1 -21920.423,E2 -21920.423} C_VEL
LIN {X 0,Y 225.88,Z 449.062,A -85,B 0,C 180,E1 -21921.517,E2 -21921.517} C_VEL
LIN {X 0,Y 227.787,Z 436.226,A -85,B 0,C 180,E1 -21922.374,E2 -21922.374} C_VEL
LIN {X 0,Y 229.017,Z 422.864,A -85,B 0,C 180,E1 -21922.929,E2 -21922.929} C_VEL
LIN {X 0,Y 231.359,Z 385.492,A -85,B 0,C 180,E1 -21923.987,E2 -21923.987} C_VEL
LIN {X 0,Y 225.589,Z 373.432,A -85,B 0,C 180,E1 -21926.092,E2 -21926.092} C_VEL
LIN {X 0,Y 221.054,Z 365.337,A -85,B 0,C 180,E1 -21927.823,E2 -21927.823} C_VEL
LIN {X 0,Y 214.259,Z 355.016,A -85,B 0,C 180,E1 -21930.602,E2 -21930.602} C_VEL
LIN {X 0,Y 208.205,Z 346.68,A -85,B 0,C 180,E1 -21933.365,E2 -21933.365} C_VEL
LIN {X 0,Y 205.45,Z 342.93,A -85,B 0,C 180,E1 -21934.744,E2 -21934.744} C_VEL
LIN {X 0,Y 202.177,Z 339.056,A -85,B 0,C 180,E1 -21936.464,E2 -21936.464} C_VEL
LIN {X 0,Y 201.204,Z 337.449,A -85,B 0,C 180,E1 -21937.035,E2 -21937.035} C_VEL
LIN {X 0,Y 198.672,Z 335.081,A -85,B 0,C 180,E1 -21938.468,E2 -21938.468} C_VEL
LIN {X 0,Y 197.108,Z 332.214,A -85,B 0,C 180,E1 -21939.52,E2 -21939.52} C_VEL
LIN {X 0,Y 194.532,Z 330.404,A -85,B 0,C 180,E1 -21941.135,E2 -21941.135} C_VEL
LIN {X 0,Y 193.023,Z 327.762,A -85,B 0,C 180,E1 -21942.285,E2 -21942.285} C_VEL
LIN {X 0,Y 192.752,Z 326.467,A -85,B 0,C 180,E1 -21942.63,E2 -21942.63} C_VEL
LIN {X 0,Y 192.856,Z 326.456,A -85,B 0,C 180,E1 -21947.37,E2 -21947.37} C_VEL
LIN {X 0,Y 193.072,Z 326.421,A -85,B 0,C 180,E1 -21951.628,E2 -21951.628} C_VEL
LIN {X 0,Y 193.265,Z 326.408,A -85,B 0,C 180,E1 -21957.916,E2 -21957.916} C_VEL
LIN {X 0,Y 193.443,Z 326.37,A -85,B 0,C 180,E1 -21960,E2 -21960} C_VEL
LIN {X 0,Y 192.98,Z 326.439,A -85,B 0,C 180,E1 -21964.177,E2 -21964.177} C_VEL
LIN {X 0,Y 193.082,Z 326.429,A -85,B 0,C 180,E1 -21968.372,E2 -21968.372} C_VEL
LIN {X 0,Y 193.014,Z 326.423,A -85,B 0,C 180,E1 -21970.538,E2 -21970.538} C_VEL
LIN {X 0,Y 192.76,Z 326.457,A -85,B 0,C 180,E1 -21976.958,E2 -21976.958} C_VEL
LIN {X 0,Y 192.619,Z 326.476,A -85,B 0,C 180,E1 -21981.399,E2 -21981.399} C_VEL
LIN {X 0,Y 192.65,Z 326.481,A -85,B 0,C 180,E1 -21984.213,E2 -21984.213} C_VEL
LIN {X 0,Y 192.703,Z 326.648,A -85,B 0,C 180,E1 -21988.302,E2 -21988.302} C_VEL
LIN {X 0,Y 193.907,Z 330.225,A -85,B 0,C 180,E1 -21992.01,E2 -21992.01} C_VEL
LIN {X 0,Y 197.317,Z 335.124,A -85,B 0,C 180,E1 -21994.355,E2 -21994.355} C_VEL
LIN {X 0,Y 199.264,Z 337.525,A -85,B 0,C 180,E1 -21995.555,E2 -21995.555} C_VEL
